PROPERTY boPin261_48XSFaultToolValue : BOOL
GET
                    boPin261_48XSFaultToolValue := boPin261_48XSFault.Value;

                  
END_GET
END_PROPERTY

PROPERTY boPin254_48XSFaultToolValue : BOOL
GET
                    boPin254_48XSFaultToolValue := boPin254_48XSFault.Value;

                  
END_GET
END_PROPERTY

PROPERTY boPin260_48XSFaultToolValue : BOOL
GET
                    boPin260_48XSFaultToolValue := boPin260_48XSFault.Value;

                  
END_GET
END_PROPERTY

PROPERTY boPin253_48XSFaultToolValue : BOOL
GET
                    boPin253_48XSFaultToolValue := boPin253_48XSFault.Value;

                  
END_GET
END_PROPERTY

PROPERTY boPin270_48XSFaultToolValue : BOOL
GET
                    boPin270_48XSFaultToolValue := boPin270_48XSFault.Value;

                  
END_GET
END_PROPERTY

PROPERTY boPin276_48XSFaultToolValue : BOOL
GET
                    boPin276_48XSFaultToolValue := boPin276_48XSFault.Value;

                  
END_GET
END_PROPERTY

PROPERTY boPin277_48XSFaultToolValue : BOOL
GET
                    boPin277_48XSFaultToolValue := boPin277_48XSFault.Value;

                  
END_GET
END_PROPERTY

PROPERTY boPin275_48XSFaultToolValue : BOOL
GET
                    boPin275_48XSFaultToolValue := boPin275_48XSFault.Value;

                  
END_GET
END_PROPERTY

PROPERTY boPin268_48XSFaultToolValue : BOOL
GET
                    boPin268_48XSFaultToolValue := boPin268_48XSFault.Value;

                  
END_GET
END_PROPERTY

PROPERTY boPin274_48XSFaultToolValue : BOOL
GET
                    boPin274_48XSFaultToolValue := boPin274_48XSFault.Value;

                  
END_GET
END_PROPERTY

PROPERTY boPin267_48XSFaultToolValue : BOOL
GET
                    boPin267_48XSFaultToolValue := boPin267_48XSFault.Value;

                  
END_GET
END_PROPERTY

METHOD InitializeCanSignals
                  boPin136_48XSFault.AppScalingDivisor :=1;
boPin136_48XSFault.AppScalingMultiplier :=1;
boPin136_48XSFault.AppScalingOffset :=0;
boPin136_48XSFault.AppUnit :="";
boPin136_48XSFault.CanDefault :=0;
boPin136_48XSFault.CanInit :=0;
boPin136_48XSFault.CanMax :=1;
boPin136_48XSFault.CanMin :=0;
boPin136_48XSFault.CanUnit :="";
boPin136_48XSFault.Description :="for the Neotec diag pages";
boPin136_48XSFault.ErrorReaction := eErrorReaction.ERSIG_DFLT;
boPin136_48XSFault.ReceiverAdress :=1;
boPin136_48XSFault.ToolScalingDivisor :=1;
boPin136_48XSFault.ToolScalingMultiplier :=1;
boPin136_48XSFault.ToolScalingOffset :=0;
boPin136_48XSFault.ToolUnit :="";

boPin148_48XSFault.AppScalingDivisor :=1;
boPin148_48XSFault.AppScalingMultiplier :=1;
boPin148_48XSFault.AppScalingOffset :=0;
boPin148_48XSFault.AppUnit :="";
boPin148_48XSFault.CanDefault :=0;
boPin148_48XSFault.CanInit :=0;
boPin148_48XSFault.CanMax :=1;
boPin148_48XSFault.CanMin :=0;
boPin148_48XSFault.CanUnit :="";
boPin148_48XSFault.Description :="for the Neotec diag pages";
boPin148_48XSFault.ErrorReaction := eErrorReaction.ERSIG_DFLT;
boPin148_48XSFault.ReceiverAdress :=1;
boPin148_48XSFault.ToolScalingDivisor :=1;
boPin148_48XSFault.ToolScalingMultiplier :=1;
boPin148_48XSFault.ToolScalingOffset :=0;
boPin148_48XSFault.ToolUnit :="";

boPin135_48XSFault.AppScalingDivisor :=1;
boPin135_48XSFault.AppScalingMultiplier :=1;
boPin135_48XSFault.AppScalingOffset :=0;
boPin135_48XSFault.AppUnit :="";
boPin135_48XSFault.CanDefault :=0;
boPin135_48XSFault.CanInit :=0;
boPin135_48XSFault.CanMax :=1;
boPin135_48XSFault.CanMin :=0;
boPin135_48XSFault.CanUnit :="";
boPin135_48XSFault.Description :="for the Neotec diag pages";
boPin135_48XSFault.ErrorReaction := eErrorReaction.ERSIG_DFLT;
boPin135_48XSFault.ReceiverAdress :=1;
boPin135_48XSFault.ToolScalingDivisor :=1;
boPin135_48XSFault.ToolScalingMultiplier :=1;
boPin135_48XSFault.ToolScalingOffset :=0;
boPin135_48XSFault.ToolUnit :="";

boPin147_48XSFault.AppScalingDivisor :=1;
boPin147_48XSFault.AppScalingMultiplier :=1;
boPin147_48XSFault.AppScalingOffset :=0;
boPin147_48XSFault.AppUnit :="";
boPin147_48XSFault.CanDefault :=0;
boPin147_48XSFault.CanInit :=0;
boPin147_48XSFault.CanMax :=1;
boPin147_48XSFault.CanMin :=0;
boPin147_48XSFault.CanUnit :="";
boPin147_48XSFault.Description :="for the Neotec diag pages";
boPin147_48XSFault.ErrorReaction := eErrorReaction.ERSIG_DFLT;
boPin147_48XSFault.ReceiverAdress :=1;
boPin147_48XSFault.ToolScalingDivisor :=1;
boPin147_48XSFault.ToolScalingMultiplier :=1;
boPin147_48XSFault.ToolScalingOffset :=0;
boPin147_48XSFault.ToolUnit :="";

boPin269_48XSFault.AppScalingDivisor :=1;
boPin269_48XSFault.AppScalingMultiplier :=1;
boPin269_48XSFault.AppScalingOffset :=0;
boPin269_48XSFault.AppUnit :="";
boPin269_48XSFault.CanDefault :=0;
boPin269_48XSFault.CanInit :=0;
boPin269_48XSFault.CanMax :=1;
boPin269_48XSFault.CanMin :=0;
boPin269_48XSFault.CanUnit :="";
boPin269_48XSFault.Description :="for the Neotec diag pages";
boPin269_48XSFault.ErrorReaction := eErrorReaction.ERSIG_DFLT;
boPin269_48XSFault.ReceiverAdress :=1;
boPin269_48XSFault.ToolScalingDivisor :=1;
boPin269_48XSFault.ToolScalingMultiplier :=1;
boPin269_48XSFault.ToolScalingOffset :=0;
boPin269_48XSFault.ToolUnit :="";

boPin118_48XSFault.AppScalingDivisor :=1;
boPin118_48XSFault.AppScalingMultiplier :=1;
boPin118_48XSFault.AppScalingOffset :=0;
boPin118_48XSFault.AppUnit :="";
boPin118_48XSFault.CanDefault :=0;
boPin118_48XSFault.CanInit :=0;
boPin118_48XSFault.CanMax :=1;
boPin118_48XSFault.CanMin :=0;
boPin118_48XSFault.CanUnit :="";
boPin118_48XSFault.Description :="for the Neotec diag pages";
boPin118_48XSFault.ErrorReaction := eErrorReaction.ERSIG_DFLT;
boPin118_48XSFault.ReceiverAdress :=1;
boPin118_48XSFault.ToolScalingDivisor :=1;
boPin118_48XSFault.ToolScalingMultiplier :=1;
boPin118_48XSFault.ToolScalingOffset :=0;
boPin118_48XSFault.ToolUnit :="";

boPin106_48XSFault.AppScalingDivisor :=1;
boPin106_48XSFault.AppScalingMultiplier :=1;
boPin106_48XSFault.AppScalingOffset :=0;
boPin106_48XSFault.AppUnit :="";
boPin106_48XSFault.CanDefault :=0;
boPin106_48XSFault.CanInit :=0;
boPin106_48XSFault.CanMax :=1;
boPin106_48XSFault.CanMin :=0;
boPin106_48XSFault.CanUnit :="";
boPin106_48XSFault.Description :="for the Neotec diag pages";
boPin106_48XSFault.ErrorReaction := eErrorReaction.ERSIG_DFLT;
boPin106_48XSFault.ReceiverAdress :=1;
boPin106_48XSFault.ToolScalingDivisor :=1;
boPin106_48XSFault.ToolScalingMultiplier :=1;
boPin106_48XSFault.ToolScalingOffset :=0;
boPin106_48XSFault.ToolUnit :="";

boPin117_48XSFault.AppScalingDivisor :=1;
boPin117_48XSFault.AppScalingMultiplier :=1;
boPin117_48XSFault.AppScalingOffset :=0;
boPin117_48XSFault.AppUnit :="";
boPin117_48XSFault.CanDefault :=0;
boPin117_48XSFault.CanInit :=0;
boPin117_48XSFault.CanMax :=1;
boPin117_48XSFault.CanMin :=0;
boPin117_48XSFault.CanUnit :="";
boPin117_48XSFault.Description :="for the Neotec diag pages";
boPin117_48XSFault.ErrorReaction := eErrorReaction.ERSIG_DFLT;
boPin117_48XSFault.ReceiverAdress :=1;
boPin117_48XSFault.ToolScalingDivisor :=1;
boPin117_48XSFault.ToolScalingMultiplier :=1;
boPin117_48XSFault.ToolScalingOffset :=0;
boPin117_48XSFault.ToolUnit :="";

boPin105_48XSFault.AppScalingDivisor :=1;
boPin105_48XSFault.AppScalingMultiplier :=1;
boPin105_48XSFault.AppScalingOffset :=0;
boPin105_48XSFault.AppUnit :="";
boPin105_48XSFault.CanDefault :=0;
boPin105_48XSFault.CanInit :=0;
boPin105_48XSFault.CanMax :=1;
boPin105_48XSFault.CanMin :=0;
boPin105_48XSFault.CanUnit :="";
boPin105_48XSFault.Description :="for the Neotec diag pages";
boPin105_48XSFault.ErrorReaction := eErrorReaction.ERSIG_DFLT;
boPin105_48XSFault.ReceiverAdress :=1;
boPin105_48XSFault.ToolScalingDivisor :=1;
boPin105_48XSFault.ToolScalingMultiplier :=1;
boPin105_48XSFault.ToolScalingOffset :=0;
boPin105_48XSFault.ToolUnit :="";

boPin116_48XSFault.AppScalingDivisor :=1;
boPin116_48XSFault.AppScalingMultiplier :=1;
boPin116_48XSFault.AppScalingOffset :=0;
boPin116_48XSFault.AppUnit :="";
boPin116_48XSFault.CanDefault :=0;
boPin116_48XSFault.CanInit :=0;
boPin116_48XSFault.CanMax :=1;
boPin116_48XSFault.CanMin :=0;
boPin116_48XSFault.CanUnit :="";
boPin116_48XSFault.Description :="for the Neotec diag pages";
boPin116_48XSFault.ErrorReaction := eErrorReaction.ERSIG_DFLT;
boPin116_48XSFault.ReceiverAdress :=1;
boPin116_48XSFault.ToolScalingDivisor :=1;
boPin116_48XSFault.ToolScalingMultiplier :=1;
boPin116_48XSFault.ToolScalingOffset :=0;
boPin116_48XSFault.ToolUnit :="";

boPin104_48XSFault.AppScalingDivisor :=1;
boPin104_48XSFault.AppScalingMultiplier :=1;
boPin104_48XSFault.AppScalingOffset :=0;
boPin104_48XSFault.AppUnit :="";
boPin104_48XSFault.CanDefault :=0;
boPin104_48XSFault.CanInit :=0;
boPin104_48XSFault.CanMax :=1;
boPin104_48XSFault.CanMin :=0;
boPin104_48XSFault.CanUnit :="";
boPin104_48XSFault.Description :="for the Neotec diag pages";
boPin104_48XSFault.ErrorReaction := eErrorReaction.ERSIG_DFLT;
boPin104_48XSFault.ReceiverAdress :=1;
boPin104_48XSFault.ToolScalingDivisor :=1;
boPin104_48XSFault.ToolScalingMultiplier :=1;
boPin104_48XSFault.ToolScalingOffset :=0;
boPin104_48XSFault.ToolUnit :="";

boPin115_48XSFault.AppScalingDivisor :=1;
boPin115_48XSFault.AppScalingMultiplier :=1;
boPin115_48XSFault.AppScalingOffset :=0;
boPin115_48XSFault.AppUnit :="";
boPin115_48XSFault.CanDefault :=0;
boPin115_48XSFault.CanInit :=0;
boPin115_48XSFault.CanMax :=1;
boPin115_48XSFault.CanMin :=0;
boPin115_48XSFault.CanUnit :="";
boPin115_48XSFault.Description :="for the Neotec diag pages";
boPin115_48XSFault.ErrorReaction := eErrorReaction.ERSIG_DFLT;
boPin115_48XSFault.ReceiverAdress :=1;
boPin115_48XSFault.ToolScalingDivisor :=1;
boPin115_48XSFault.ToolScalingMultiplier :=1;
boPin115_48XSFault.ToolScalingOffset :=0;
boPin115_48XSFault.ToolUnit :="";

boPin103_48XSFault.AppScalingDivisor :=1;
boPin103_48XSFault.AppScalingMultiplier :=1;
boPin103_48XSFault.AppScalingOffset :=0;
boPin103_48XSFault.AppUnit :="";
boPin103_48XSFault.CanDefault :=0;
boPin103_48XSFault.CanInit :=0;
boPin103_48XSFault.CanMax :=1;
boPin103_48XSFault.CanMin :=0;
boPin103_48XSFault.CanUnit :="";
boPin103_48XSFault.Description :="for the Neotec diag pages";
boPin103_48XSFault.ErrorReaction := eErrorReaction.ERSIG_DFLT;
boPin103_48XSFault.ReceiverAdress :=1;
boPin103_48XSFault.ToolScalingDivisor :=1;
boPin103_48XSFault.ToolScalingMultiplier :=1;
boPin103_48XSFault.ToolScalingOffset :=0;
boPin103_48XSFault.ToolUnit :="";

boPin120_48XSFault.AppScalingDivisor :=1;
boPin120_48XSFault.AppScalingMultiplier :=1;
boPin120_48XSFault.AppScalingOffset :=0;
boPin120_48XSFault.AppUnit :="";
boPin120_48XSFault.CanDefault :=0;
boPin120_48XSFault.CanInit :=0;
boPin120_48XSFault.CanMax :=1;
boPin120_48XSFault.CanMin :=0;
boPin120_48XSFault.CanUnit :="";
boPin120_48XSFault.Description :="for the Neotec diag pages";
boPin120_48XSFault.ErrorReaction := eErrorReaction.ERSIG_DFLT;
boPin120_48XSFault.ReceiverAdress :=1;
boPin120_48XSFault.ToolScalingDivisor :=1;
boPin120_48XSFault.ToolScalingMultiplier :=1;
boPin120_48XSFault.ToolScalingOffset :=0;
boPin120_48XSFault.ToolUnit :="";

boPin108_48XSFault.AppScalingDivisor :=1;
boPin108_48XSFault.AppScalingMultiplier :=1;
boPin108_48XSFault.AppScalingOffset :=0;
boPin108_48XSFault.AppUnit :="";
boPin108_48XSFault.CanDefault :=0;
boPin108_48XSFault.CanInit :=0;
boPin108_48XSFault.CanMax :=1;
boPin108_48XSFault.CanMin :=0;
boPin108_48XSFault.CanUnit :="";
boPin108_48XSFault.Description :="for the Neotec diag pages";
boPin108_48XSFault.ErrorReaction := eErrorReaction.ERSIG_DFLT;
boPin108_48XSFault.ReceiverAdress :=1;
boPin108_48XSFault.ToolScalingDivisor :=1;
boPin108_48XSFault.ToolScalingMultiplier :=1;
boPin108_48XSFault.ToolScalingOffset :=0;
boPin108_48XSFault.ToolUnit :="";

boPin119_48XSFault.AppScalingDivisor :=1;
boPin119_48XSFault.AppScalingMultiplier :=1;
boPin119_48XSFault.AppScalingOffset :=0;
boPin119_48XSFault.AppUnit :="";
boPin119_48XSFault.CanDefault :=0;
boPin119_48XSFault.CanInit :=0;
boPin119_48XSFault.CanMax :=1;
boPin119_48XSFault.CanMin :=0;
boPin119_48XSFault.CanUnit :="";
boPin119_48XSFault.Description :="for the Neotec diag pages";
boPin119_48XSFault.ErrorReaction := eErrorReaction.ERSIG_DFLT;
boPin119_48XSFault.ReceiverAdress :=1;
boPin119_48XSFault.ToolScalingDivisor :=1;
boPin119_48XSFault.ToolScalingMultiplier :=1;
boPin119_48XSFault.ToolScalingOffset :=0;
boPin119_48XSFault.ToolUnit :="";

boPin107_48XSFault.AppScalingDivisor :=1;
boPin107_48XSFault.AppScalingMultiplier :=1;
boPin107_48XSFault.AppScalingOffset :=0;
boPin107_48XSFault.AppUnit :="";
boPin107_48XSFault.CanDefault :=0;
boPin107_48XSFault.CanInit :=0;
boPin107_48XSFault.CanMax :=1;
boPin107_48XSFault.CanMin :=0;
boPin107_48XSFault.CanUnit :="";
boPin107_48XSFault.Description :="for the Neotec diag pages";
boPin107_48XSFault.ErrorReaction := eErrorReaction.ERSIG_DFLT;
boPin107_48XSFault.ReceiverAdress :=1;
boPin107_48XSFault.ToolScalingDivisor :=1;
boPin107_48XSFault.ToolScalingMultiplier :=1;
boPin107_48XSFault.ToolScalingOffset :=0;
boPin107_48XSFault.ToolUnit :="";

boPin144_48XSFault.AppScalingDivisor :=1;
boPin144_48XSFault.AppScalingMultiplier :=1;
boPin144_48XSFault.AppScalingOffset :=0;
boPin144_48XSFault.AppUnit :="";
boPin144_48XSFault.CanDefault :=0;
boPin144_48XSFault.CanInit :=0;
boPin144_48XSFault.CanMax :=1;
boPin144_48XSFault.CanMin :=0;
boPin144_48XSFault.CanUnit :="";
boPin144_48XSFault.Description :="for the Neotec diag pages";
boPin144_48XSFault.ErrorReaction := eErrorReaction.ERSIG_DFLT;
boPin144_48XSFault.ReceiverAdress :=1;
boPin144_48XSFault.ToolScalingDivisor :=1;
boPin144_48XSFault.ToolScalingMultiplier :=1;
boPin144_48XSFault.ToolScalingOffset :=0;
boPin144_48XSFault.ToolUnit :="";

boPin132_48XSFault.AppScalingDivisor :=1;
boPin132_48XSFault.AppScalingMultiplier :=1;
boPin132_48XSFault.AppScalingOffset :=0;
boPin132_48XSFault.AppUnit :="";
boPin132_48XSFault.CanDefault :=0;
boPin132_48XSFault.CanInit :=0;
boPin132_48XSFault.CanMax :=1;
boPin132_48XSFault.CanMin :=0;
boPin132_48XSFault.CanUnit :="";
boPin132_48XSFault.Description :="for the Neotec diag pages";
boPin132_48XSFault.ErrorReaction := eErrorReaction.ERSIG_DFLT;
boPin132_48XSFault.ReceiverAdress :=1;
boPin132_48XSFault.ToolScalingDivisor :=1;
boPin132_48XSFault.ToolScalingMultiplier :=1;
boPin132_48XSFault.ToolScalingOffset :=0;
boPin132_48XSFault.ToolUnit :="";

boPin143_48XSFault.AppScalingDivisor :=1;
boPin143_48XSFault.AppScalingMultiplier :=1;
boPin143_48XSFault.AppScalingOffset :=0;
boPin143_48XSFault.AppUnit :="";
boPin143_48XSFault.CanDefault :=0;
boPin143_48XSFault.CanInit :=0;
boPin143_48XSFault.CanMax :=1;
boPin143_48XSFault.CanMin :=0;
boPin143_48XSFault.CanUnit :="";
boPin143_48XSFault.Description :="for the Neotec diag pages";
boPin143_48XSFault.ErrorReaction := eErrorReaction.ERSIG_DFLT;
boPin143_48XSFault.ReceiverAdress :=1;
boPin143_48XSFault.ToolScalingDivisor :=1;
boPin143_48XSFault.ToolScalingMultiplier :=1;
boPin143_48XSFault.ToolScalingOffset :=0;
boPin143_48XSFault.ToolUnit :="";

boPin131_48XSFault.AppScalingDivisor :=1;
boPin131_48XSFault.AppScalingMultiplier :=1;
boPin131_48XSFault.AppScalingOffset :=0;
boPin131_48XSFault.AppUnit :="";
boPin131_48XSFault.CanDefault :=0;
boPin131_48XSFault.CanInit :=0;
boPin131_48XSFault.CanMax :=1;
boPin131_48XSFault.CanMin :=0;
boPin131_48XSFault.CanUnit :="";
boPin131_48XSFault.Description :="for the Neotec diag pages";
boPin131_48XSFault.ErrorReaction := eErrorReaction.ERSIG_DFLT;
boPin131_48XSFault.ReceiverAdress :=1;
boPin131_48XSFault.ToolScalingDivisor :=1;
boPin131_48XSFault.ToolScalingMultiplier :=1;
boPin131_48XSFault.ToolScalingOffset :=0;
boPin131_48XSFault.ToolUnit :="";

boPin142_48XSFault.AppScalingDivisor :=1;
boPin142_48XSFault.AppScalingMultiplier :=1;
boPin142_48XSFault.AppScalingOffset :=0;
boPin142_48XSFault.AppUnit :="";
boPin142_48XSFault.CanDefault :=0;
boPin142_48XSFault.CanInit :=0;
boPin142_48XSFault.CanMax :=1;
boPin142_48XSFault.CanMin :=0;
boPin142_48XSFault.CanUnit :="";
boPin142_48XSFault.Description :="for the Neotec diag pages";
boPin142_48XSFault.ErrorReaction := eErrorReaction.ERSIG_DFLT;
boPin142_48XSFault.ReceiverAdress :=1;
boPin142_48XSFault.ToolScalingDivisor :=1;
boPin142_48XSFault.ToolScalingMultiplier :=1;
boPin142_48XSFault.ToolScalingOffset :=0;
boPin142_48XSFault.ToolUnit :="";

boPin130_48XSFault.AppScalingDivisor :=1;
boPin130_48XSFault.AppScalingMultiplier :=1;
boPin130_48XSFault.AppScalingOffset :=0;
boPin130_48XSFault.AppUnit :="";
boPin130_48XSFault.CanDefault :=0;
boPin130_48XSFault.CanInit :=0;
boPin130_48XSFault.CanMax :=1;
boPin130_48XSFault.CanMin :=0;
boPin130_48XSFault.CanUnit :="";
boPin130_48XSFault.Description :="for the Neotec diag pages";
boPin130_48XSFault.ErrorReaction := eErrorReaction.ERSIG_DFLT;
boPin130_48XSFault.ReceiverAdress :=1;
boPin130_48XSFault.ToolScalingDivisor :=1;
boPin130_48XSFault.ToolScalingMultiplier :=1;
boPin130_48XSFault.ToolScalingOffset :=0;
boPin130_48XSFault.ToolUnit :="";

boPin141_48XSFault.AppScalingDivisor :=1;
boPin141_48XSFault.AppScalingMultiplier :=1;
boPin141_48XSFault.AppScalingOffset :=0;
boPin141_48XSFault.AppUnit :="";
boPin141_48XSFault.CanDefault :=0;
boPin141_48XSFault.CanInit :=0;
boPin141_48XSFault.CanMax :=1;
boPin141_48XSFault.CanMin :=0;
boPin141_48XSFault.CanUnit :="";
boPin141_48XSFault.Description :="for the Neotec diag pages";
boPin141_48XSFault.ErrorReaction := eErrorReaction.ERSIG_DFLT;
boPin141_48XSFault.ReceiverAdress :=1;
boPin141_48XSFault.ToolScalingDivisor :=1;
boPin141_48XSFault.ToolScalingMultiplier :=1;
boPin141_48XSFault.ToolScalingOffset :=0;
boPin141_48XSFault.ToolUnit :="";

boPin129_48XSFault.AppScalingDivisor :=1;
boPin129_48XSFault.AppScalingMultiplier :=1;
boPin129_48XSFault.AppScalingOffset :=0;
boPin129_48XSFault.AppUnit :="";
boPin129_48XSFault.CanDefault :=0;
boPin129_48XSFault.CanInit :=0;
boPin129_48XSFault.CanMax :=1;
boPin129_48XSFault.CanMin :=0;
boPin129_48XSFault.CanUnit :="";
boPin129_48XSFault.Description :="for the Neotec diag pages";
boPin129_48XSFault.ErrorReaction := eErrorReaction.ERSIG_DFLT;
boPin129_48XSFault.ReceiverAdress :=1;
boPin129_48XSFault.ToolScalingDivisor :=1;
boPin129_48XSFault.ToolScalingMultiplier :=1;
boPin129_48XSFault.ToolScalingOffset :=0;
boPin129_48XSFault.ToolUnit :="";

boPin152_48XSFault.AppScalingDivisor :=1;
boPin152_48XSFault.AppScalingMultiplier :=1;
boPin152_48XSFault.AppScalingOffset :=0;
boPin152_48XSFault.AppUnit :="";
boPin152_48XSFault.CanDefault :=0;
boPin152_48XSFault.CanInit :=0;
boPin152_48XSFault.CanMax :=1;
boPin152_48XSFault.CanMin :=0;
boPin152_48XSFault.CanUnit :="";
boPin152_48XSFault.Description :="for the Neotec diag pages";
boPin152_48XSFault.ErrorReaction := eErrorReaction.ERSIG_DFLT;
boPin152_48XSFault.ReceiverAdress :=1;
boPin152_48XSFault.ToolScalingDivisor :=1;
boPin152_48XSFault.ToolScalingMultiplier :=1;
boPin152_48XSFault.ToolScalingOffset :=0;
boPin152_48XSFault.ToolUnit :="";

boPin140_48XSFault.AppScalingDivisor :=1;
boPin140_48XSFault.AppScalingMultiplier :=1;
boPin140_48XSFault.AppScalingOffset :=0;
boPin140_48XSFault.AppUnit :="";
boPin140_48XSFault.CanDefault :=0;
boPin140_48XSFault.CanInit :=0;
boPin140_48XSFault.CanMax :=1;
boPin140_48XSFault.CanMin :=0;
boPin140_48XSFault.CanUnit :="";
boPin140_48XSFault.Description :="for the Neotec diag pages";
boPin140_48XSFault.ErrorReaction := eErrorReaction.ERSIG_DFLT;
boPin140_48XSFault.ReceiverAdress :=1;
boPin140_48XSFault.ToolScalingDivisor :=1;
boPin140_48XSFault.ToolScalingMultiplier :=1;
boPin140_48XSFault.ToolScalingOffset :=0;
boPin140_48XSFault.ToolUnit :="";

boPin151_48XSFault.AppScalingDivisor :=1;
boPin151_48XSFault.AppScalingMultiplier :=1;
boPin151_48XSFault.AppScalingOffset :=0;
boPin151_48XSFault.AppUnit :="";
boPin151_48XSFault.CanDefault :=0;
boPin151_48XSFault.CanInit :=0;
boPin151_48XSFault.CanMax :=1;
boPin151_48XSFault.CanMin :=0;
boPin151_48XSFault.CanUnit :="";
boPin151_48XSFault.Description :="for the Neotec diag pages";
boPin151_48XSFault.ErrorReaction := eErrorReaction.ERSIG_DFLT;
boPin151_48XSFault.ReceiverAdress :=1;
boPin151_48XSFault.ToolScalingDivisor :=1;
boPin151_48XSFault.ToolScalingMultiplier :=1;
boPin151_48XSFault.ToolScalingOffset :=0;
boPin151_48XSFault.ToolUnit :="";

boPin139_48XSFault.AppScalingDivisor :=1;
boPin139_48XSFault.AppScalingMultiplier :=1;
boPin139_48XSFault.AppScalingOffset :=0;
boPin139_48XSFault.AppUnit :="";
boPin139_48XSFault.CanDefault :=0;
boPin139_48XSFault.CanInit :=0;
boPin139_48XSFault.CanMax :=1;
boPin139_48XSFault.CanMin :=0;
boPin139_48XSFault.CanUnit :="";
boPin139_48XSFault.Description :="for the Neotec diag pages";
boPin139_48XSFault.ErrorReaction := eErrorReaction.ERSIG_DFLT;
boPin139_48XSFault.ReceiverAdress :=1;
boPin139_48XSFault.ToolScalingDivisor :=1;
boPin139_48XSFault.ToolScalingMultiplier :=1;
boPin139_48XSFault.ToolScalingOffset :=0;
boPin139_48XSFault.ToolUnit :="";

boPin150_48XSFault.AppScalingDivisor :=1;
boPin150_48XSFault.AppScalingMultiplier :=1;
boPin150_48XSFault.AppScalingOffset :=0;
boPin150_48XSFault.AppUnit :="";
boPin150_48XSFault.CanDefault :=0;
boPin150_48XSFault.CanInit :=0;
boPin150_48XSFault.CanMax :=1;
boPin150_48XSFault.CanMin :=0;
boPin150_48XSFault.CanUnit :="";
boPin150_48XSFault.Description :="for the Neotec diag pages";
boPin150_48XSFault.ErrorReaction := eErrorReaction.ERSIG_DFLT;
boPin150_48XSFault.ReceiverAdress :=1;
boPin150_48XSFault.ToolScalingDivisor :=1;
boPin150_48XSFault.ToolScalingMultiplier :=1;
boPin150_48XSFault.ToolScalingOffset :=0;
boPin150_48XSFault.ToolUnit :="";

boPin138_48XSFault.AppScalingDivisor :=1;
boPin138_48XSFault.AppScalingMultiplier :=1;
boPin138_48XSFault.AppScalingOffset :=0;
boPin138_48XSFault.AppUnit :="";
boPin138_48XSFault.CanDefault :=0;
boPin138_48XSFault.CanInit :=0;
boPin138_48XSFault.CanMax :=1;
boPin138_48XSFault.CanMin :=0;
boPin138_48XSFault.CanUnit :="";
boPin138_48XSFault.Description :="for the Neotec diag pages";
boPin138_48XSFault.ErrorReaction := eErrorReaction.ERSIG_DFLT;
boPin138_48XSFault.ReceiverAdress :=1;
boPin138_48XSFault.ToolScalingDivisor :=1;
boPin138_48XSFault.ToolScalingMultiplier :=1;
boPin138_48XSFault.ToolScalingOffset :=0;
boPin138_48XSFault.ToolUnit :="";

boPin149_48XSFault.AppScalingDivisor :=1;
boPin149_48XSFault.AppScalingMultiplier :=1;
boPin149_48XSFault.AppScalingOffset :=0;
boPin149_48XSFault.AppUnit :="";
boPin149_48XSFault.CanDefault :=0;
boPin149_48XSFault.CanInit :=0;
boPin149_48XSFault.CanMax :=1;
boPin149_48XSFault.CanMin :=0;
boPin149_48XSFault.CanUnit :="";
boPin149_48XSFault.Description :="for the Neotec diag pages";
boPin149_48XSFault.ErrorReaction := eErrorReaction.ERSIG_DFLT;
boPin149_48XSFault.ReceiverAdress :=1;
boPin149_48XSFault.ToolScalingDivisor :=1;
boPin149_48XSFault.ToolScalingMultiplier :=1;
boPin149_48XSFault.ToolScalingOffset :=0;
boPin149_48XSFault.ToolUnit :="";

boPin137_48XSFault.AppScalingDivisor :=1;
boPin137_48XSFault.AppScalingMultiplier :=1;
boPin137_48XSFault.AppScalingOffset :=0;
boPin137_48XSFault.AppUnit :="";
boPin137_48XSFault.CanDefault :=0;
boPin137_48XSFault.CanInit :=0;
boPin137_48XSFault.CanMax :=1;
boPin137_48XSFault.CanMin :=0;
boPin137_48XSFault.CanUnit :="";
boPin137_48XSFault.Description :="for the Neotec diag pages";
boPin137_48XSFault.ErrorReaction := eErrorReaction.ERSIG_DFLT;
boPin137_48XSFault.ReceiverAdress :=1;
boPin137_48XSFault.ToolScalingDivisor :=1;
boPin137_48XSFault.ToolScalingMultiplier :=1;
boPin137_48XSFault.ToolScalingOffset :=0;
boPin137_48XSFault.ToolUnit :="";

boPin126_48XSFault.AppScalingDivisor :=1;
boPin126_48XSFault.AppScalingMultiplier :=1;
boPin126_48XSFault.AppScalingOffset :=0;
boPin126_48XSFault.AppUnit :="";
boPin126_48XSFault.CanDefault :=0;
boPin126_48XSFault.CanInit :=0;
boPin126_48XSFault.CanMax :=1;
boPin126_48XSFault.CanMin :=0;
boPin126_48XSFault.CanUnit :="";
boPin126_48XSFault.Description :="for the Neotec diag pages";
boPin126_48XSFault.ErrorReaction := eErrorReaction.ERSIG_DFLT;
boPin126_48XSFault.ReceiverAdress :=1;
boPin126_48XSFault.ToolScalingDivisor :=1;
boPin126_48XSFault.ToolScalingMultiplier :=1;
boPin126_48XSFault.ToolScalingOffset :=0;
boPin126_48XSFault.ToolUnit :="";

boPin114_48XSFault.AppScalingDivisor :=1;
boPin114_48XSFault.AppScalingMultiplier :=1;
boPin114_48XSFault.AppScalingOffset :=0;
boPin114_48XSFault.AppUnit :="";
boPin114_48XSFault.CanDefault :=0;
boPin114_48XSFault.CanInit :=0;
boPin114_48XSFault.CanMax :=1;
boPin114_48XSFault.CanMin :=0;
boPin114_48XSFault.CanUnit :="";
boPin114_48XSFault.Description :="for the Neotec diag pages";
boPin114_48XSFault.ErrorReaction := eErrorReaction.ERSIG_DFLT;
boPin114_48XSFault.ReceiverAdress :=1;
boPin114_48XSFault.ToolScalingDivisor :=1;
boPin114_48XSFault.ToolScalingMultiplier :=1;
boPin114_48XSFault.ToolScalingOffset :=0;
boPin114_48XSFault.ToolUnit :="";

boPin125_48XSFault.AppScalingDivisor :=1;
boPin125_48XSFault.AppScalingMultiplier :=1;
boPin125_48XSFault.AppScalingOffset :=0;
boPin125_48XSFault.AppUnit :="";
boPin125_48XSFault.CanDefault :=0;
boPin125_48XSFault.CanInit :=0;
boPin125_48XSFault.CanMax :=1;
boPin125_48XSFault.CanMin :=0;
boPin125_48XSFault.CanUnit :="";
boPin125_48XSFault.Description :="for the Neotec diag pages";
boPin125_48XSFault.ErrorReaction := eErrorReaction.ERSIG_DFLT;
boPin125_48XSFault.ReceiverAdress :=1;
boPin125_48XSFault.ToolScalingDivisor :=1;
boPin125_48XSFault.ToolScalingMultiplier :=1;
boPin125_48XSFault.ToolScalingOffset :=0;
boPin125_48XSFault.ToolUnit :="";

boPin113_48XSFault.AppScalingDivisor :=1;
boPin113_48XSFault.AppScalingMultiplier :=1;
boPin113_48XSFault.AppScalingOffset :=0;
boPin113_48XSFault.AppUnit :="";
boPin113_48XSFault.CanDefault :=0;
boPin113_48XSFault.CanInit :=0;
boPin113_48XSFault.CanMax :=1;
boPin113_48XSFault.CanMin :=0;
boPin113_48XSFault.CanUnit :="";
boPin113_48XSFault.Description :="for the Neotec diag pages";
boPin113_48XSFault.ErrorReaction := eErrorReaction.ERSIG_DFLT;
boPin113_48XSFault.ReceiverAdress :=1;
boPin113_48XSFault.ToolScalingDivisor :=1;
boPin113_48XSFault.ToolScalingMultiplier :=1;
boPin113_48XSFault.ToolScalingOffset :=0;
boPin113_48XSFault.ToolUnit :="";

boPin124_48XSFault.AppScalingDivisor :=1;
boPin124_48XSFault.AppScalingMultiplier :=1;
boPin124_48XSFault.AppScalingOffset :=0;
boPin124_48XSFault.AppUnit :="";
boPin124_48XSFault.CanDefault :=0;
boPin124_48XSFault.CanInit :=0;
boPin124_48XSFault.CanMax :=1;
boPin124_48XSFault.CanMin :=0;
boPin124_48XSFault.CanUnit :="";
boPin124_48XSFault.Description :="for the Neotec diag pages";
boPin124_48XSFault.ErrorReaction := eErrorReaction.ERSIG_DFLT;
boPin124_48XSFault.ReceiverAdress :=1;
boPin124_48XSFault.ToolScalingDivisor :=1;
boPin124_48XSFault.ToolScalingMultiplier :=1;
boPin124_48XSFault.ToolScalingOffset :=0;
boPin124_48XSFault.ToolUnit :="";

boPin112_48XSFault.AppScalingDivisor :=1;
boPin112_48XSFault.AppScalingMultiplier :=1;
boPin112_48XSFault.AppScalingOffset :=0;
boPin112_48XSFault.AppUnit :="";
boPin112_48XSFault.CanDefault :=0;
boPin112_48XSFault.CanInit :=0;
boPin112_48XSFault.CanMax :=1;
boPin112_48XSFault.CanMin :=0;
boPin112_48XSFault.CanUnit :="";
boPin112_48XSFault.Description :="for the Neotec diag pages";
boPin112_48XSFault.ErrorReaction := eErrorReaction.ERSIG_DFLT;
boPin112_48XSFault.ReceiverAdress :=1;
boPin112_48XSFault.ToolScalingDivisor :=1;
boPin112_48XSFault.ToolScalingMultiplier :=1;
boPin112_48XSFault.ToolScalingOffset :=0;
boPin112_48XSFault.ToolUnit :="";

boPin123_48XSFault.AppScalingDivisor :=1;
boPin123_48XSFault.AppScalingMultiplier :=1;
boPin123_48XSFault.AppScalingOffset :=0;
boPin123_48XSFault.AppUnit :="";
boPin123_48XSFault.CanDefault :=0;
boPin123_48XSFault.CanInit :=0;
boPin123_48XSFault.CanMax :=1;
boPin123_48XSFault.CanMin :=0;
boPin123_48XSFault.CanUnit :="";
boPin123_48XSFault.Description :="for the Neotec diag pages";
boPin123_48XSFault.ErrorReaction := eErrorReaction.ERSIG_DFLT;
boPin123_48XSFault.ReceiverAdress :=1;
boPin123_48XSFault.ToolScalingDivisor :=1;
boPin123_48XSFault.ToolScalingMultiplier :=1;
boPin123_48XSFault.ToolScalingOffset :=0;
boPin123_48XSFault.ToolUnit :="";

boPin111_48XSFault.AppScalingDivisor :=1;
boPin111_48XSFault.AppScalingMultiplier :=1;
boPin111_48XSFault.AppScalingOffset :=0;
boPin111_48XSFault.AppUnit :="";
boPin111_48XSFault.CanDefault :=0;
boPin111_48XSFault.CanInit :=0;
boPin111_48XSFault.CanMax :=1;
boPin111_48XSFault.CanMin :=0;
boPin111_48XSFault.CanUnit :="";
boPin111_48XSFault.Description :="for the Neotec diag pages";
boPin111_48XSFault.ErrorReaction := eErrorReaction.ERSIG_DFLT;
boPin111_48XSFault.ReceiverAdress :=1;
boPin111_48XSFault.ToolScalingDivisor :=1;
boPin111_48XSFault.ToolScalingMultiplier :=1;
boPin111_48XSFault.ToolScalingOffset :=0;
boPin111_48XSFault.ToolUnit :="";

boPin133_48XSFault.AppScalingDivisor :=1;
boPin133_48XSFault.AppScalingMultiplier :=1;
boPin133_48XSFault.AppScalingOffset :=0;
boPin133_48XSFault.AppUnit :="";
boPin133_48XSFault.CanDefault :=0;
boPin133_48XSFault.CanInit :=0;
boPin133_48XSFault.CanMax :=1;
boPin133_48XSFault.CanMin :=0;
boPin133_48XSFault.CanUnit :="";
boPin133_48XSFault.Description :="for the Neotec diag pages";
boPin133_48XSFault.ErrorReaction := eErrorReaction.ERSIG_DFLT;
boPin133_48XSFault.ReceiverAdress :=1;
boPin133_48XSFault.ToolScalingDivisor :=1;
boPin133_48XSFault.ToolScalingMultiplier :=1;
boPin133_48XSFault.ToolScalingOffset :=0;
boPin133_48XSFault.ToolUnit :="";

boPin134_48XSFault.AppScalingDivisor :=1;
boPin134_48XSFault.AppScalingMultiplier :=1;
boPin134_48XSFault.AppScalingOffset :=0;
boPin134_48XSFault.AppUnit :="";
boPin134_48XSFault.CanDefault :=0;
boPin134_48XSFault.CanInit :=0;
boPin134_48XSFault.CanMax :=1;
boPin134_48XSFault.CanMin :=0;
boPin134_48XSFault.CanUnit :="";
boPin134_48XSFault.Description :="for the Neotec diag pages";
boPin134_48XSFault.ErrorReaction := eErrorReaction.ERSIG_DFLT;
boPin134_48XSFault.ReceiverAdress :=1;
boPin134_48XSFault.ToolScalingDivisor :=1;
boPin134_48XSFault.ToolScalingMultiplier :=1;
boPin134_48XSFault.ToolScalingOffset :=0;
boPin134_48XSFault.ToolUnit :="";

boPin145_48XSFault.AppScalingDivisor :=1;
boPin145_48XSFault.AppScalingMultiplier :=1;
boPin145_48XSFault.AppScalingOffset :=0;
boPin145_48XSFault.AppUnit :="";
boPin145_48XSFault.CanDefault :=0;
boPin145_48XSFault.CanInit :=0;
boPin145_48XSFault.CanMax :=1;
boPin145_48XSFault.CanMin :=0;
boPin145_48XSFault.CanUnit :="";
boPin145_48XSFault.Description :="for the Neotec diag pages";
boPin145_48XSFault.ErrorReaction := eErrorReaction.ERSIG_DFLT;
boPin145_48XSFault.ReceiverAdress :=1;
boPin145_48XSFault.ToolScalingDivisor :=1;
boPin145_48XSFault.ToolScalingMultiplier :=1;
boPin145_48XSFault.ToolScalingOffset :=0;
boPin145_48XSFault.ToolUnit :="";

boPin146_48XSFault.AppScalingDivisor :=1;
boPin146_48XSFault.AppScalingMultiplier :=1;
boPin146_48XSFault.AppScalingOffset :=0;
boPin146_48XSFault.AppUnit :="";
boPin146_48XSFault.CanDefault :=0;
boPin146_48XSFault.CanInit :=0;
boPin146_48XSFault.CanMax :=1;
boPin146_48XSFault.CanMin :=0;
boPin146_48XSFault.CanUnit :="";
boPin146_48XSFault.Description :="for the Neotec diag pages";
boPin146_48XSFault.ErrorReaction := eErrorReaction.ERSIG_DFLT;
boPin146_48XSFault.ReceiverAdress :=1;
boPin146_48XSFault.ToolScalingDivisor :=1;
boPin146_48XSFault.ToolScalingMultiplier :=1;
boPin146_48XSFault.ToolScalingOffset :=0;
boPin146_48XSFault.ToolUnit :="";

boPin263_48XSFault.AppScalingDivisor :=1;
boPin263_48XSFault.AppScalingMultiplier :=1;
boPin263_48XSFault.AppScalingOffset :=0;
boPin263_48XSFault.AppUnit :="";
boPin263_48XSFault.CanDefault :=0;
boPin263_48XSFault.CanInit :=0;
boPin263_48XSFault.CanMax :=1;
boPin263_48XSFault.CanMin :=0;
boPin263_48XSFault.CanUnit :="";
boPin263_48XSFault.Description :="for the Neotec diag pages";
boPin263_48XSFault.ErrorReaction := eErrorReaction.ERSIG_DFLT;
boPin263_48XSFault.ReceiverAdress :=1;
boPin263_48XSFault.ToolScalingDivisor :=1;
boPin263_48XSFault.ToolScalingMultiplier :=1;
boPin263_48XSFault.ToolScalingOffset :=0;
boPin263_48XSFault.ToolUnit :="";

boPin256_48XSFault.AppScalingDivisor :=1;
boPin256_48XSFault.AppScalingMultiplier :=1;
boPin256_48XSFault.AppScalingOffset :=0;
boPin256_48XSFault.AppUnit :="";
boPin256_48XSFault.CanDefault :=0;
boPin256_48XSFault.CanInit :=0;
boPin256_48XSFault.CanMax :=1;
boPin256_48XSFault.CanMin :=0;
boPin256_48XSFault.CanUnit :="";
boPin256_48XSFault.Description :="for the Neotec diag pages";
boPin256_48XSFault.ErrorReaction := eErrorReaction.ERSIG_DFLT;
boPin256_48XSFault.ReceiverAdress :=1;
boPin256_48XSFault.ToolScalingDivisor :=1;
boPin256_48XSFault.ToolScalingMultiplier :=1;
boPin256_48XSFault.ToolScalingOffset :=0;
boPin256_48XSFault.ToolUnit :="";

boPin262_48XSFault.AppScalingDivisor :=1;
boPin262_48XSFault.AppScalingMultiplier :=1;
boPin262_48XSFault.AppScalingOffset :=0;
boPin262_48XSFault.AppUnit :="";
boPin262_48XSFault.CanDefault :=0;
boPin262_48XSFault.CanInit :=0;
boPin262_48XSFault.CanMax :=1;
boPin262_48XSFault.CanMin :=0;
boPin262_48XSFault.CanUnit :="";
boPin262_48XSFault.Description :="for the Neotec diag pages";
boPin262_48XSFault.ErrorReaction := eErrorReaction.ERSIG_DFLT;
boPin262_48XSFault.ReceiverAdress :=1;
boPin262_48XSFault.ToolScalingDivisor :=1;
boPin262_48XSFault.ToolScalingMultiplier :=1;
boPin262_48XSFault.ToolScalingOffset :=0;
boPin262_48XSFault.ToolUnit :="";

boPin255_48XSFault.AppScalingDivisor :=1;
boPin255_48XSFault.AppScalingMultiplier :=1;
boPin255_48XSFault.AppScalingOffset :=0;
boPin255_48XSFault.AppUnit :="";
boPin255_48XSFault.CanDefault :=0;
boPin255_48XSFault.CanInit :=0;
boPin255_48XSFault.CanMax :=1;
boPin255_48XSFault.CanMin :=0;
boPin255_48XSFault.CanUnit :="";
boPin255_48XSFault.Description :="for the Neotec diag pages";
boPin255_48XSFault.ErrorReaction := eErrorReaction.ERSIG_DFLT;
boPin255_48XSFault.ReceiverAdress :=1;
boPin255_48XSFault.ToolScalingDivisor :=1;
boPin255_48XSFault.ToolScalingMultiplier :=1;
boPin255_48XSFault.ToolScalingOffset :=0;
boPin255_48XSFault.ToolUnit :="";

boPin261_48XSFault.AppScalingDivisor :=1;
boPin261_48XSFault.AppScalingMultiplier :=1;
boPin261_48XSFault.AppScalingOffset :=0;
boPin261_48XSFault.AppUnit :="";
boPin261_48XSFault.CanDefault :=0;
boPin261_48XSFault.CanInit :=0;
boPin261_48XSFault.CanMax :=1;
boPin261_48XSFault.CanMin :=0;
boPin261_48XSFault.CanUnit :="";
boPin261_48XSFault.Description :="for the Neotec diag pages";
boPin261_48XSFault.ErrorReaction := eErrorReaction.ERSIG_DFLT;
boPin261_48XSFault.ReceiverAdress :=1;
boPin261_48XSFault.ToolScalingDivisor :=1;
boPin261_48XSFault.ToolScalingMultiplier :=1;
boPin261_48XSFault.ToolScalingOffset :=0;
boPin261_48XSFault.ToolUnit :="";

boPin254_48XSFault.AppScalingDivisor :=1;
boPin254_48XSFault.AppScalingMultiplier :=1;
boPin254_48XSFault.AppScalingOffset :=0;
boPin254_48XSFault.AppUnit :="";
boPin254_48XSFault.CanDefault :=0;
boPin254_48XSFault.CanInit :=0;
boPin254_48XSFault.CanMax :=1;
boPin254_48XSFault.CanMin :=0;
boPin254_48XSFault.CanUnit :="";
boPin254_48XSFault.Description :="for the Neotec diag pages";
boPin254_48XSFault.ErrorReaction := eErrorReaction.ERSIG_DFLT;
boPin254_48XSFault.ReceiverAdress :=1;
boPin254_48XSFault.ToolScalingDivisor :=1;
boPin254_48XSFault.ToolScalingMultiplier :=1;
boPin254_48XSFault.ToolScalingOffset :=0;
boPin254_48XSFault.ToolUnit :="";

boPin260_48XSFault.AppScalingDivisor :=1;
boPin260_48XSFault.AppScalingMultiplier :=1;
boPin260_48XSFault.AppScalingOffset :=0;
boPin260_48XSFault.AppUnit :="";
boPin260_48XSFault.CanDefault :=0;
boPin260_48XSFault.CanInit :=0;
boPin260_48XSFault.CanMax :=1;
boPin260_48XSFault.CanMin :=0;
boPin260_48XSFault.CanUnit :="";
boPin260_48XSFault.Description :="for the Neotec diag pages";
boPin260_48XSFault.ErrorReaction := eErrorReaction.ERSIG_DFLT;
boPin260_48XSFault.ReceiverAdress :=1;
boPin260_48XSFault.ToolScalingDivisor :=1;
boPin260_48XSFault.ToolScalingMultiplier :=1;
boPin260_48XSFault.ToolScalingOffset :=0;
boPin260_48XSFault.ToolUnit :="";

boPin253_48XSFault.AppScalingDivisor :=1;
boPin253_48XSFault.AppScalingMultiplier :=1;
boPin253_48XSFault.AppScalingOffset :=0;
boPin253_48XSFault.AppUnit :="";
boPin253_48XSFault.CanDefault :=0;
boPin253_48XSFault.CanInit :=0;
boPin253_48XSFault.CanMax :=1;
boPin253_48XSFault.CanMin :=0;
boPin253_48XSFault.CanUnit :="";
boPin253_48XSFault.Description :="for the Neotec diag pages";
boPin253_48XSFault.ErrorReaction := eErrorReaction.ERSIG_DFLT;
boPin253_48XSFault.ReceiverAdress :=1;
boPin253_48XSFault.ToolScalingDivisor :=1;
boPin253_48XSFault.ToolScalingMultiplier :=1;
boPin253_48XSFault.ToolScalingOffset :=0;
boPin253_48XSFault.ToolUnit :="";

boPin270_48XSFault.AppScalingDivisor :=1;
boPin270_48XSFault.AppScalingMultiplier :=1;
boPin270_48XSFault.AppScalingOffset :=0;
boPin270_48XSFault.AppUnit :="";
boPin270_48XSFault.CanDefault :=0;
boPin270_48XSFault.CanInit :=0;
boPin270_48XSFault.CanMax :=1;
boPin270_48XSFault.CanMin :=0;
boPin270_48XSFault.CanUnit :="";
boPin270_48XSFault.Description :="for the Neotec diag pages";
boPin270_48XSFault.ErrorReaction := eErrorReaction.ERSIG_DFLT;
boPin270_48XSFault.ReceiverAdress :=1;
boPin270_48XSFault.ToolScalingDivisor :=1;
boPin270_48XSFault.ToolScalingMultiplier :=1;
boPin270_48XSFault.ToolScalingOffset :=0;
boPin270_48XSFault.ToolUnit :="";

boPin276_48XSFault.AppScalingDivisor :=1;
boPin276_48XSFault.AppScalingMultiplier :=1;
boPin276_48XSFault.AppScalingOffset :=0;
boPin276_48XSFault.AppUnit :="";
boPin276_48XSFault.CanDefault :=0;
boPin276_48XSFault.CanInit :=0;
boPin276_48XSFault.CanMax :=1;
boPin276_48XSFault.CanMin :=0;
boPin276_48XSFault.CanUnit :="";
boPin276_48XSFault.Description :="for the Neotec diag pages";
boPin276_48XSFault.ErrorReaction := eErrorReaction.ERSIG_DFLT;
boPin276_48XSFault.ReceiverAdress :=1;
boPin276_48XSFault.ToolScalingDivisor :=1;
boPin276_48XSFault.ToolScalingMultiplier :=1;
boPin276_48XSFault.ToolScalingOffset :=0;
boPin276_48XSFault.ToolUnit :="";

boPin277_48XSFault.AppScalingDivisor :=1;
boPin277_48XSFault.AppScalingMultiplier :=1;
boPin277_48XSFault.AppScalingOffset :=0;
boPin277_48XSFault.AppUnit :="";
boPin277_48XSFault.CanDefault :=0;
boPin277_48XSFault.CanInit :=0;
boPin277_48XSFault.CanMax :=1;
boPin277_48XSFault.CanMin :=0;
boPin277_48XSFault.CanUnit :="";
boPin277_48XSFault.Description :="for the Neotec diag pages";
boPin277_48XSFault.ErrorReaction := eErrorReaction.ERSIG_DFLT;
boPin277_48XSFault.ReceiverAdress :=1;
boPin277_48XSFault.ToolScalingDivisor :=1;
boPin277_48XSFault.ToolScalingMultiplier :=1;
boPin277_48XSFault.ToolScalingOffset :=0;
boPin277_48XSFault.ToolUnit :="";

boPin275_48XSFault.AppScalingDivisor :=1;
boPin275_48XSFault.AppScalingMultiplier :=1;
boPin275_48XSFault.AppScalingOffset :=0;
boPin275_48XSFault.AppUnit :="";
boPin275_48XSFault.CanDefault :=0;
boPin275_48XSFault.CanInit :=0;
boPin275_48XSFault.CanMax :=1;
boPin275_48XSFault.CanMin :=0;
boPin275_48XSFault.CanUnit :="";
boPin275_48XSFault.Description :="for the Neotec diag pages";
boPin275_48XSFault.ErrorReaction := eErrorReaction.ERSIG_DFLT;
boPin275_48XSFault.ReceiverAdress :=1;
boPin275_48XSFault.ToolScalingDivisor :=1;
boPin275_48XSFault.ToolScalingMultiplier :=1;
boPin275_48XSFault.ToolScalingOffset :=0;
boPin275_48XSFault.ToolUnit :="";

boPin268_48XSFault.AppScalingDivisor :=1;
boPin268_48XSFault.AppScalingMultiplier :=1;
boPin268_48XSFault.AppScalingOffset :=0;
boPin268_48XSFault.AppUnit :="";
boPin268_48XSFault.CanDefault :=0;
boPin268_48XSFault.CanInit :=0;
boPin268_48XSFault.CanMax :=1;
boPin268_48XSFault.CanMin :=0;
boPin268_48XSFault.CanUnit :="";
boPin268_48XSFault.Description :="for the Neotec diag pages";
boPin268_48XSFault.ErrorReaction := eErrorReaction.ERSIG_DFLT;
boPin268_48XSFault.ReceiverAdress :=1;
boPin268_48XSFault.ToolScalingDivisor :=1;
boPin268_48XSFault.ToolScalingMultiplier :=1;
boPin268_48XSFault.ToolScalingOffset :=0;
boPin268_48XSFault.ToolUnit :="";

boPin274_48XSFault.AppScalingDivisor :=1;
boPin274_48XSFault.AppScalingMultiplier :=1;
boPin274_48XSFault.AppScalingOffset :=0;
boPin274_48XSFault.AppUnit :="";
boPin274_48XSFault.CanDefault :=0;
boPin274_48XSFault.CanInit :=0;
boPin274_48XSFault.CanMax :=1;
boPin274_48XSFault.CanMin :=0;
boPin274_48XSFault.CanUnit :="";
boPin274_48XSFault.Description :="for the Neotec diag pages";
boPin274_48XSFault.ErrorReaction := eErrorReaction.ERSIG_DFLT;
boPin274_48XSFault.ReceiverAdress :=1;
boPin274_48XSFault.ToolScalingDivisor :=1;
boPin274_48XSFault.ToolScalingMultiplier :=1;
boPin274_48XSFault.ToolScalingOffset :=0;
boPin274_48XSFault.ToolUnit :="";

boPin267_48XSFault.AppScalingDivisor :=1;
boPin267_48XSFault.AppScalingMultiplier :=1;
boPin267_48XSFault.AppScalingOffset :=0;
boPin267_48XSFault.AppUnit :="";
boPin267_48XSFault.CanDefault :=0;
boPin267_48XSFault.CanInit :=0;
boPin267_48XSFault.CanMax :=1;
boPin267_48XSFault.CanMin :=0;
boPin267_48XSFault.CanUnit :="";
boPin267_48XSFault.Description :="for the Neotec diag pages";
boPin267_48XSFault.ErrorReaction := eErrorReaction.ERSIG_DFLT;
boPin267_48XSFault.ReceiverAdress :=1;
boPin267_48XSFault.ToolScalingDivisor :=1;
boPin267_48XSFault.ToolScalingMultiplier :=1;
boPin267_48XSFault.ToolScalingOffset :=0;
boPin267_48XSFault.ToolUnit :="";


                
END_METHOD
END_FUNCTION_BLOCK

FUNCTION_BLOCK Msg9C0SendToEvision7MessageClass EXTENDS CanReceiveMessageClass
  VAR_INPUT
    boPin144_48XS : BoolCanSignalClass;
    boPin132_48XS : BoolCanSignalClass;
    boPin143_48XS : BoolCanSignalClass;
    boPin131_48XS : BoolCanSignalClass;
    boPin142_48XS : BoolCanSignalClass;
    boPin130_48XS : BoolCanSignalClass;
    boPin141_48XS : BoolCanSignalClass;
    boPin129_48XS : BoolCanSignalClass;
    boPin152_48XS : BoolCanSignalClass;
    boPin140_48XS : BoolCanSignalClass;
    boPin151_48XS : BoolCanSignalClass;
    boPin139_48XS : BoolCanSignalClass;
    boPin150_48XS : BoolCanSignalClass;
    boPin138_48XS : BoolCanSignalClass;
    boPin149_48XS : BoolCanSignalClass;
    boPin263_48XS : BoolCanSignalClass;
    boPin256_48XS : BoolCanSignalClass;
    boPin262_48XS : BoolCanSignalClass;
    boPin255_48XS : BoolCanSignalClass;
    boPin261_48XS : BoolCanSignalClass;
    boPin254_48XS : BoolCanSignalClass;
    boPin260_48XS : BoolCanSignalClass;
    boPin253_48XS : BoolCanSignalClass;
    boPin275_48XS : BoolCanSignalClass;
    boPin268_48XS : BoolCanSignalClass;
    boPin274_48XS : BoolCanSignalClass;
    boPin267_48XS : BoolCanSignalClass;
    i16gPressureBrakeSensorValue : Int16CanSignalClass;
    u8gLightsMode : UInt8CanSignalClass;
    bogOsciServiceBrakinBrakeOn : BoolCanSignalClass;
    bogFixeServiceBrakinBrakeOn : BoolCanSignalClass;
    bogBothServiceBrakinBrakeOn : BoolCanSignalClass;
    bogActiveWhiteLights15746 : BoolCanSignalClass;
    Counter : UInt32CanSignalClass;
  END_VAR

            
          

METHOD SetData
  VAR_INPUT
    CanMsgPointer : POINTER TO CanMessageClass;
  END_VAR
                  IF IsValidPointer(canMsgPointer,'SetData') THEN
	SUPER^.SetData(CanMsgPointer);
	//Set the new data
	boPin144_48XS.Value := canMsgPointer^.GetBoolOnBit(0);
	boPin132_48XS.Value := canMsgPointer^.GetBoolOnBit(1);
	boPin143_48XS.Value := canMsgPointer^.GetBoolOnBit(2);
	boPin131_48XS.Value := canMsgPointer^.GetBoolOnBit(3);
	boPin142_48XS.Value := canMsgPointer^.GetBoolOnBit(4);
	boPin130_48XS.Value := canMsgPointer^.GetBoolOnBit(5);
	boPin141_48XS.Value := canMsgPointer^.GetBoolOnBit(6);
	boPin129_48XS.Value := canMsgPointer^.GetBoolOnBit(7);
	boPin152_48XS.Value := canMsgPointer^.GetBoolOnBit(8);
	boPin140_48XS.Value := canMsgPointer^.GetBoolOnBit(9);
	boPin151_48XS.Value := canMsgPointer^.GetBoolOnBit(10);
	boPin139_48XS.Value := canMsgPointer^.GetBoolOnBit(11);
	boPin150_48XS.Value := canMsgPointer^.GetBoolOnBit(12);
	boPin138_48XS.Value := canMsgPointer^.GetBoolOnBit(13);
	boPin149_48XS.Value := canMsgPointer^.GetBoolOnBit(14);
	boPin263_48XS.Value := canMsgPointer^.GetBoolOnBit(15);
	boPin256_48XS.Value := canMsgPointer^.GetBoolOnBit(16);
	boPin262_48XS.Value := canMsgPointer^.GetBoolOnBit(17);
	boPin255_48XS.Value := canMsgPointer^.GetBoolOnBit(18);
	boPin261_48XS.Value := canMsgPointer^.GetBoolOnBit(19);
	boPin254_48XS.Value := canMsgPointer^.GetBoolOnBit(20);
	boPin260_48XS.Value := canMsgPointer^.GetBoolOnBit(21);
	boPin253_48XS.Value := canMsgPointer^.GetBoolOnBit(22);
	boPin275_48XS.Value := canMsgPointer^.GetBoolOnBit(23);
	boPin268_48XS.Value := canMsgPointer^.GetBoolOnBit(24);
	boPin274_48XS.Value := canMsgPointer^.GetBoolOnBit(25);
	boPin267_48XS.Value := canMsgPointer^.GetBoolOnBit(26);
	i16gPressureBrakeSensorValue.Value := canMsgPointer^.GetInt16(32);
	u8gLightsMode.Value := canMsgPointer^.GetUint8(48);
	bogOsciServiceBrakinBrakeOn.Value := canMsgPointer^.GetBoolOnBit(56);
	bogFixeServiceBrakinBrakeOn.Value := canMsgPointer^.GetBoolOnBit(57);
	bogBothServiceBrakinBrakeOn.Value := canMsgPointer^.GetBoolOnBit(58);
	bogActiveWhiteLights15746.Value := canMsgPointer^.GetBoolOnBit(59);
	//And increase the counter
	Counter.Value := CanMsgPointer^.Counter.Value;
END_IF

                
END_METHOD

PROPERTY boPin144_48XSRawValue : BOOL
GET
                    boPin144_48XSRawValue := boPin144_48XS.Value;

                  
END_GET
END_PROPERTY

PROPERTY boPin132_48XSRawValue : BOOL
GET
                    boPin132_48XSRawValue := boPin132_48XS.Value;

                  
END_GET
END_PROPERTY

PROPERTY boPin143_48XSRawValue : BOOL
GET
                    boPin143_48XSRawValue := boPin143_48XS.Value;

                  
END_GET
END_PROPERTY

PROPERTY boPin131_48XSRawValue : BOOL
GET
                    boPin131_48XSRawValue := boPin131_48XS.Value;

                  
END_GET
END_PROPERTY

PROPERTY boPin142_48XSRawValue : BOOL
GET
                    boPin142_48XSRawValue := boPin142_48XS.Value;

                  
END_GET
END_PROPERTY

PROPERTY boPin130_48XSRawValue : BOOL
GET
                    boPin130_48XSRawValue := boPin130_48XS.Value;

                  
END_GET
END_PROPERTY

PROPERTY boPin141_48XSRawValue : BOOL
GET
                    boPin141_48XSRawValue := boPin141_48XS.Value;

                  
END_GET
END_PROPERTY

PROPERTY boPin129_48XSRawValue : BOOL
GET
                    boPin129_48XSRawValue := boPin129_48XS.Value;

                  
END_GET
END_PROPERTY

PROPERTY boPin152_48XSRawValue : BOOL
GET
                    boPin152_48XSRawValue := boPin152_48XS.Value;

                  
END_GET
END_PROPERTY

PROPERTY boPin140_48XSRawValue : BOOL
GET
                    boPin140_48XSRawValue := boPin140_48XS.Value;

                  
END_GET
END_PROPERTY

PROPERTY boPin151_48XSRawValue : BOOL
GET
                    boPin151_48XSRawValue := boPin151_48XS.Value;

                  
END_GET
END_PROPERTY

PROPERTY boPin139_48XSRawValue : BOOL
GET
                    boPin139_48XSRawValue := boPin139_48XS.Value;

                  
END_GET
END_PROPERTY

PROPERTY boPin150_48XSRawValue : BOOL
GET
                    boPin150_48XSRawValue := boPin150_48XS.Value;

                  
END_GET
END_PROPERTY

PROPERTY boPin138_48XSRawValue : BOOL
GET
                    boPin138_48XSRawValue := boPin138_48XS.Value;

                  
END_GET
END_PROPERTY

PROPERTY boPin149_48XSRawValue : BOOL
GET
                    boPin149_48XSRawValue := boPin149_48XS.Value;

                  
END_GET
END_PROPERTY

PROPERTY boPin263_48XSRawValue : BOOL
GET
                    boPin263_48XSRawValue := boPin263_48XS.Value;

                  
END_GET
END_PROPERTY

PROPERTY boPin256_48XSRawValue : BOOL
GET
                    boPin256_48XSRawValue := boPin256_48XS.Value;

                  
END_GET
END_PROPERTY

PROPERTY boPin262_48XSRawValue : BOOL
GET
                    boPin262_48XSRawValue := boPin262_48XS.Value;

                  
END_GET
END_PROPERTY

PROPERTY boPin255_48XSRawValue : BOOL
GET
                    boPin255_48XSRawValue := boPin255_48XS.Value;

                  
END_GET
END_PROPERTY

PROPERTY boPin261_48XSRawValue : BOOL
GET
                    boPin261_48XSRawValue := boPin261_48XS.Value;

                  
END_GET
END_PROPERTY

PROPERTY boPin254_48XSRawValue : BOOL
GET
                    boPin254_48XSRawValue := boPin254_48XS.Value;

                  
END_GET
END_PROPERTY

PROPERTY boPin260_48XSRawValue : BOOL
GET
                    boPin260_48XSRawValue := boPin260_48XS.Value;

                  
END_GET
END_PROPERTY

PROPERTY boPin253_48XSRawValue : BOOL
GET
                    boPin253_48XSRawValue := boPin253_48XS.Value;

                  
END_GET
END_PROPERTY

PROPERTY boPin275_48XSRawValue : BOOL
GET
                    boPin275_48XSRawValue := boPin275_48XS.Value;

                  
END_GET
END_PROPERTY

PROPERTY boPin268_48XSRawValue : BOOL
GET
                    boPin268_48XSRawValue := boPin268_48XS.Value;

                  
END_GET
END_PROPERTY

PROPERTY boPin274_48XSRawValue : BOOL
GET
                    boPin274_48XSRawValue := boPin274_48XS.Value;

                  
END_GET
END_PROPERTY

PROPERTY boPin267_48XSRawValue : BOOL
GET
                    boPin267_48XSRawValue := boPin267_48XS.Value;

                  
END_GET
END_PROPERTY

PROPERTY i16gPressureBrakeSensorValueRawValue : INT
GET
                    IF i16gPressureBrakeSensorValue.AppScalingMultiplier = 0 THEN
	_MatchLog^.Error("Get i16gPressureBrakeSensorValueRawValue", "Division by Zero!");
	RETURN;
End_IF

i16gPressureBrakeSensorValueRawValue := TO_INT((i16gPressureBrakeSensorValue.Value - i16gPressureBrakeSensorValue.AppScalingOffset) * i16gPressureBrakeSensorValue.AppScalingDivisor / i16gPressureBrakeSensorValue.AppScalingMultiplier);

                  
END_GET
END_PROPERTY

PROPERTY u8gLightsModeRawValue : USINT
GET
                    IF u8gLightsMode.AppScalingMultiplier = 0 THEN
	_MatchLog^.Error("Get u8gLightsModeRawValue", "Division by Zero!");
	RETURN;
End_IF

u8gLightsModeRawValue := TO_USINT((u8gLightsMode.Value - u8gLightsMode.AppScalingOffset) * u8gLightsMode.AppScalingDivisor / u8gLightsMode.AppScalingMultiplier);

                  
END_GET
END_PROPERTY

PROPERTY bogOsciServiceBrakinBrakeOnRawValue : BOOL
GET
                    bogOsciServiceBrakinBrakeOnRawValue := bogOsciServiceBrakinBrakeOn.Value;

                  
END_GET
END_PROPERTY

PROPERTY bogFixeServiceBrakinBrakeOnRawValue : BOOL
GET
                    bogFixeServiceBrakinBrakeOnRawValue := bogFixeServiceBrakinBrakeOn.Value;

                  
END_GET
END_PROPERTY

PROPERTY bogBothServiceBrakinBrakeOnRawValue : BOOL
GET
                    bogBothServiceBrakinBrakeOnRawValue := bogBothServiceBrakinBrakeOn.Value;

                  
END_GET
END_PROPERTY

PROPERTY bogActiveWhiteLights15746RawValue : BOOL
GET
                    bogActiveWhiteLights15746RawValue := bogActiveWhiteLights15746.Value;

                  
END_GET
END_PROPERTY

PROPERTY boPin144_48XSToolValue : BOOL
GET
                    boPin144_48XSToolValue := boPin144_48XS.Value;

                  
END_GET
END_PROPERTY

PROPERTY boPin132_48XSToolValue : BOOL
GET
                    boPin132_48XSToolValue := boPin132_48XS.Value;

                  
END_GET
END_PROPERTY

PROPERTY boPin143_48XSToolValue : BOOL
GET
                    boPin143_48XSToolValue := boPin143_48XS.Value;

                  
END_GET
END_PROPERTY

PROPERTY boPin131_48XSToolValue : BOOL
GET
                    boPin131_48XSToolValue := boPin131_48XS.Value;

                  
END_GET
END_PROPERTY

PROPERTY boPin142_48XSToolValue : BOOL
GET
                    boPin142_48XSToolValue := boPin142_48XS.Value;

                  
END_GET
END_PROPERTY

PROPERTY boPin130_48XSToolValue : BOOL
GET
                    boPin130_48XSToolValue := boPin130_48XS.Value;

                  
END_GET
END_PROPERTY

PROPERTY boPin141_48XSToolValue : BOOL
GET
                    boPin141_48XSToolValue := boPin141_48XS.Value;

                  
END_GET
END_PROPERTY

PROPERTY boPin129_48XSToolValue : BOOL
GET
                    boPin129_48XSToolValue := boPin129_48XS.Value;

                  
END_GET
END_PROPERTY

PROPERTY boPin152_48XSToolValue : BOOL
GET
                    boPin152_48XSToolValue := boPin152_48XS.Value;

                  
END_GET
END_PROPERTY

PROPERTY boPin140_48XSToolValue : BOOL
GET
                    boPin140_48XSToolValue := boPin140_48XS.Value;

                  
END_GET
END_PROPERTY

PROPERTY boPin151_48XSToolValue : BOOL
GET
                    boPin151_48XSToolValue := boPin151_48XS.Value;

                  
END_GET
END_PROPERTY

PROPERTY boPin139_48XSToolValue : BOOL
GET
                    boPin139_48XSToolValue := boPin139_48XS.Value;

                  
END_GET
END_PROPERTY

PROPERTY boPin150_48XSToolValue : BOOL
GET
                    boPin150_48XSToolValue := boPin150_48XS.Value;

                  
END_GET
END_PROPERTY

PROPERTY boPin138_48XSToolValue : BOOL
GET
                    boPin138_48XSToolValue := boPin138_48XS.Value;

                  
END_GET
END_PROPERTY

PROPERTY boPin149_48XSToolValue : BOOL
GET
                    boPin149_48XSToolValue := boPin149_48XS.Value;

                  
END_GET
END_PROPERTY

PROPERTY boPin263_48XSToolValue : BOOL
GET
                    boPin263_48XSToolValue := boPin263_48XS.Value;

                  
END_GET
END_PROPERTY

PROPERTY boPin256_48XSToolValue : BOOL
GET
                    boPin256_48XSToolValue := boPin256_48XS.Value;

                  
END_GET
END_PROPERTY

PROPERTY boPin262_48XSToolValue : BOOL
GET
                    boPin262_48XSToolValue := boPin262_48XS.Value;

                  
END_GET
END_PROPERTY

PROPERTY boPin255_48XSToolValue : BOOL
GET
                    boPin255_48XSToolValue := boPin255_48XS.Value;

                  
END_GET
END_PROPERTY

PROPERTY boPin261_48XSToolValue : BOOL
GET
                    boPin261_48XSToolValue := boPin261_48XS.Value;

                  
END_GET
END_PROPERTY

PROPERTY boPin254_48XSToolValue : BOOL
GET
                    boPin254_48XSToolValue := boPin254_48XS.Value;

                  
END_GET
END_PROPERTY

PROPERTY boPin260_48XSToolValue : BOOL
GET
                    boPin260_48XSToolValue := boPin260_48XS.Value;

                  
END_GET
END_PROPERTY

PROPERTY boPin253_48XSToolValue : BOOL
GET
                    boPin253_48XSToolValue := boPin253_48XS.Value;

                  
END_GET
END_PROPERTY

PROPERTY boPin275_48XSToolValue : BOOL
GET
                    boPin275_48XSToolValue := boPin275_48XS.Value;

                  
END_GET
END_PROPERTY

PROPERTY boPin268_48XSToolValue : BOOL
GET
                    boPin268_48XSToolValue := boPin268_48XS.Value;

                  
END_GET
END_PROPERTY

PROPERTY boPin274_48XSToolValue : BOOL
GET
                    boPin274_48XSToolValue := boPin274_48XS.Value;

                  
END_GET
END_PROPERTY

PROPERTY boPin267_48XSToolValue : BOOL
GET
                    boPin267_48XSToolValue := boPin267_48XS.Value;

                  
END_GET
END_PROPERTY

PROPERTY i16gPressureBrakeSensorValueToolValue : INT
GET
                    IF i16gPressureBrakeSensorValue.ToolScalingDivisor = 0 OR i16gPressureBrakeSensorValue.AppScalingMultiplier = 0 THEN
	_MatchLog^.Error("Get i16gPressureBrakeSensorValueToolValue", "Division by Zero!");
	RETURN;
END_IF

i16gPressureBrakeSensorValueToolValue := TO_INT(((i16gPressureBrakeSensorValue.Value - i16gPressureBrakeSensorValue.AppScalingOffset) * i16gPressureBrakeSensorValue.AppScalingDivisor / i16gPressureBrakeSensorValue.AppScalingMultiplier * i16gPressureBrakeSensorValue.ToolScalingMultiplier / i16gPressureBrakeSensorValue.ToolScalingDivisor) + i16gPressureBrakeSensorValue.ToolScalingOffset);

                  
END_GET
END_PROPERTY

PROPERTY u8gLightsModeToolValue : USINT
GET
                    IF u8gLightsMode.ToolScalingDivisor = 0 OR u8gLightsMode.AppScalingMultiplier = 0 THEN
	_MatchLog^.Error("Get u8gLightsModeToolValue", "Division by Zero!");
	RETURN;
END_IF

u8gLightsModeToolValue := TO_USINT(((u8gLightsMode.Value - u8gLightsMode.AppScalingOffset) * u8gLightsMode.AppScalingDivisor / u8gLightsMode.AppScalingMultiplier * u8gLightsMode.ToolScalingMultiplier / u8gLightsMode.ToolScalingDivisor) + u8gLightsMode.ToolScalingOffset);

                  
END_GET
END_PROPERTY

PROPERTY bogOsciServiceBrakinBrakeOnToolValue : BOOL
GET
                    bogOsciServiceBrakinBrakeOnToolValue := bogOsciServiceBrakinBrakeOn.Value;

                  
END_GET
END_PROPERTY

PROPERTY bogFixeServiceBrakinBrakeOnToolValue : BOOL
GET
                    bogFixeServiceBrakinBrakeOnToolValue := bogFixeServiceBrakinBrakeOn.Value;

                  
END_GET
END_PROPERTY

PROPERTY bogBothServiceBrakinBrakeOnToolValue : BOOL
GET
                    bogBothServiceBrakinBrakeOnToolValue := bogBothServiceBrakinBrakeOn.Value;

                  
END_GET
END_PROPERTY

PROPERTY bogActiveWhiteLights15746ToolValue : BOOL
GET
                    bogActiveWhiteLights15746ToolValue := bogActiveWhiteLights15746.Value;

                  
END_GET
END_PROPERTY

METHOD InitializeCanSignals
                  boPin144_48XS.AppScalingDivisor :=1;
boPin144_48XS.AppScalingMultiplier :=1;
boPin144_48XS.AppScalingOffset :=0;
boPin144_48XS.AppUnit :="";
boPin144_48XS.CanDefault :=0;
boPin144_48XS.CanInit :=0;
boPin144_48XS.CanMax :=1;
boPin144_48XS.CanMin :=0;
boPin144_48XS.CanUnit :="";
boPin144_48XS.Description :="for the Neotec diag pages";
boPin144_48XS.ErrorReaction := eErrorReaction.ERSIG_DFLT;
boPin144_48XS.ReceiverAdress :=1;
boPin144_48XS.ToolScalingDivisor :=1;
boPin144_48XS.ToolScalingMultiplier :=1;
boPin144_48XS.ToolScalingOffset :=0;
boPin144_48XS.ToolUnit :="";

boPin132_48XS.AppScalingDivisor :=1;
boPin132_48XS.AppScalingMultiplier :=1;
boPin132_48XS.AppScalingOffset :=0;
boPin132_48XS.AppUnit :="";
boPin132_48XS.CanDefault :=0;
boPin132_48XS.CanInit :=0;
boPin132_48XS.CanMax :=1;
boPin132_48XS.CanMin :=0;
boPin132_48XS.CanUnit :="";
boPin132_48XS.Description :="for the Neotec diag pages";
boPin132_48XS.ErrorReaction := eErrorReaction.ERSIG_DFLT;
boPin132_48XS.ReceiverAdress :=1;
boPin132_48XS.ToolScalingDivisor :=1;
boPin132_48XS.ToolScalingMultiplier :=1;
boPin132_48XS.ToolScalingOffset :=0;
boPin132_48XS.ToolUnit :="";

boPin143_48XS.AppScalingDivisor :=1;
boPin143_48XS.AppScalingMultiplier :=1;
boPin143_48XS.AppScalingOffset :=0;
boPin143_48XS.AppUnit :="";
boPin143_48XS.CanDefault :=0;
boPin143_48XS.CanInit :=0;
boPin143_48XS.CanMax :=1;
boPin143_48XS.CanMin :=0;
boPin143_48XS.CanUnit :="";
boPin143_48XS.Description :="for the Neotec diag pages";
boPin143_48XS.ErrorReaction := eErrorReaction.ERSIG_DFLT;
boPin143_48XS.ReceiverAdress :=1;
boPin143_48XS.ToolScalingDivisor :=1;
boPin143_48XS.ToolScalingMultiplier :=1;
boPin143_48XS.ToolScalingOffset :=0;
boPin143_48XS.ToolUnit :="";

boPin131_48XS.AppScalingDivisor :=1;
boPin131_48XS.AppScalingMultiplier :=1;
boPin131_48XS.AppScalingOffset :=0;
boPin131_48XS.AppUnit :="";
boPin131_48XS.CanDefault :=0;
boPin131_48XS.CanInit :=0;
boPin131_48XS.CanMax :=1;
boPin131_48XS.CanMin :=0;
boPin131_48XS.CanUnit :="";
boPin131_48XS.Description :="for the Neotec diag pages";
boPin131_48XS.ErrorReaction := eErrorReaction.ERSIG_DFLT;
boPin131_48XS.ReceiverAdress :=1;
boPin131_48XS.ToolScalingDivisor :=1;
boPin131_48XS.ToolScalingMultiplier :=1;
boPin131_48XS.ToolScalingOffset :=0;
boPin131_48XS.ToolUnit :="";

boPin142_48XS.AppScalingDivisor :=1;
boPin142_48XS.AppScalingMultiplier :=1;
boPin142_48XS.AppScalingOffset :=0;
boPin142_48XS.AppUnit :="";
boPin142_48XS.CanDefault :=0;
boPin142_48XS.CanInit :=0;
boPin142_48XS.CanMax :=1;
boPin142_48XS.CanMin :=0;
boPin142_48XS.CanUnit :="";
boPin142_48XS.Description :="for the Neotec diag pages";
boPin142_48XS.ErrorReaction := eErrorReaction.ERSIG_DFLT;
boPin142_48XS.ReceiverAdress :=1;
boPin142_48XS.ToolScalingDivisor :=1;
boPin142_48XS.ToolScalingMultiplier :=1;
boPin142_48XS.ToolScalingOffset :=0;
boPin142_48XS.ToolUnit :="";

boPin130_48XS.AppScalingDivisor :=1;
boPin130_48XS.AppScalingMultiplier :=1;
boPin130_48XS.AppScalingOffset :=0;
boPin130_48XS.AppUnit :="";
boPin130_48XS.CanDefault :=0;
boPin130_48XS.CanInit :=0;
boPin130_48XS.CanMax :=1;
boPin130_48XS.CanMin :=0;
boPin130_48XS.CanUnit :="";
boPin130_48XS.Description :="for the Neotec diag pages";
boPin130_48XS.ErrorReaction := eErrorReaction.ERSIG_DFLT;
boPin130_48XS.ReceiverAdress :=1;
boPin130_48XS.ToolScalingDivisor :=1;
boPin130_48XS.ToolScalingMultiplier :=1;
boPin130_48XS.ToolScalingOffset :=0;
boPin130_48XS.ToolUnit :="";

boPin141_48XS.AppScalingDivisor :=1;
boPin141_48XS.AppScalingMultiplier :=1;
boPin141_48XS.AppScalingOffset :=0;
boPin141_48XS.AppUnit :="";
boPin141_48XS.CanDefault :=0;
boPin141_48XS.CanInit :=0;
boPin141_48XS.CanMax :=1;
boPin141_48XS.CanMin :=0;
boPin141_48XS.CanUnit :="";
boPin141_48XS.Description :="for the Neotec diag pages";
boPin141_48XS.ErrorReaction := eErrorReaction.ERSIG_DFLT;
boPin141_48XS.ReceiverAdress :=1;
boPin141_48XS.ToolScalingDivisor :=1;
boPin141_48XS.ToolScalingMultiplier :=1;
boPin141_48XS.ToolScalingOffset :=0;
boPin141_48XS.ToolUnit :="";

boPin129_48XS.AppScalingDivisor :=1;
boPin129_48XS.AppScalingMultiplier :=1;
boPin129_48XS.AppScalingOffset :=0;
boPin129_48XS.AppUnit :="";
boPin129_48XS.CanDefault :=0;
boPin129_48XS.CanInit :=0;
boPin129_48XS.CanMax :=1;
boPin129_48XS.CanMin :=0;
boPin129_48XS.CanUnit :="";
boPin129_48XS.Description :="for the Neotec diag pages";
boPin129_48XS.ErrorReaction := eErrorReaction.ERSIG_DFLT;
boPin129_48XS.ReceiverAdress :=1;
boPin129_48XS.ToolScalingDivisor :=1;
boPin129_48XS.ToolScalingMultiplier :=1;
boPin129_48XS.ToolScalingOffset :=0;
boPin129_48XS.ToolUnit :="";

boPin152_48XS.AppScalingDivisor :=1;
boPin152_48XS.AppScalingMultiplier :=1;
boPin152_48XS.AppScalingOffset :=0;
boPin152_48XS.AppUnit :="";
boPin152_48XS.CanDefault :=0;
boPin152_48XS.CanInit :=0;
boPin152_48XS.CanMax :=1;
boPin152_48XS.CanMin :=0;
boPin152_48XS.CanUnit :="";
boPin152_48XS.Description :="for the Neotec diag pages";
boPin152_48XS.ErrorReaction := eErrorReaction.ERSIG_DFLT;
boPin152_48XS.ReceiverAdress :=1;
boPin152_48XS.ToolScalingDivisor :=1;
boPin152_48XS.ToolScalingMultiplier :=1;
boPin152_48XS.ToolScalingOffset :=0;
boPin152_48XS.ToolUnit :="";

boPin140_48XS.AppScalingDivisor :=1;
boPin140_48XS.AppScalingMultiplier :=1;
boPin140_48XS.AppScalingOffset :=0;
boPin140_48XS.AppUnit :="";
boPin140_48XS.CanDefault :=0;
boPin140_48XS.CanInit :=0;
boPin140_48XS.CanMax :=1;
boPin140_48XS.CanMin :=0;
boPin140_48XS.CanUnit :="";
boPin140_48XS.Description :="for the Neotec diag pages";
boPin140_48XS.ErrorReaction := eErrorReaction.ERSIG_DFLT;
boPin140_48XS.ReceiverAdress :=1;
boPin140_48XS.ToolScalingDivisor :=1;
boPin140_48XS.ToolScalingMultiplier :=1;
boPin140_48XS.ToolScalingOffset :=0;
boPin140_48XS.ToolUnit :="";

boPin151_48XS.AppScalingDivisor :=1;
boPin151_48XS.AppScalingMultiplier :=1;
boPin151_48XS.AppScalingOffset :=0;
boPin151_48XS.AppUnit :="";
boPin151_48XS.CanDefault :=0;
boPin151_48XS.CanInit :=0;
boPin151_48XS.CanMax :=1;
boPin151_48XS.CanMin :=0;
boPin151_48XS.CanUnit :="";
boPin151_48XS.Description :="for the Neotec diag pages";
boPin151_48XS.ErrorReaction := eErrorReaction.ERSIG_DFLT;
boPin151_48XS.ReceiverAdress :=1;
boPin151_48XS.ToolScalingDivisor :=1;
boPin151_48XS.ToolScalingMultiplier :=1;
boPin151_48XS.ToolScalingOffset :=0;
boPin151_48XS.ToolUnit :="";

boPin139_48XS.AppScalingDivisor :=1;
boPin139_48XS.AppScalingMultiplier :=1;
boPin139_48XS.AppScalingOffset :=0;
boPin139_48XS.AppUnit :="";
boPin139_48XS.CanDefault :=0;
boPin139_48XS.CanInit :=0;
boPin139_48XS.CanMax :=1;
boPin139_48XS.CanMin :=0;
boPin139_48XS.CanUnit :="";
boPin139_48XS.Description :="for the Neotec diag pages";
boPin139_48XS.ErrorReaction := eErrorReaction.ERSIG_DFLT;
boPin139_48XS.ReceiverAdress :=1;
boPin139_48XS.ToolScalingDivisor :=1;
boPin139_48XS.ToolScalingMultiplier :=1;
boPin139_48XS.ToolScalingOffset :=0;
boPin139_48XS.ToolUnit :="";

boPin150_48XS.AppScalingDivisor :=1;
boPin150_48XS.AppScalingMultiplier :=1;
boPin150_48XS.AppScalingOffset :=0;
boPin150_48XS.AppUnit :="";
boPin150_48XS.CanDefault :=0;
boPin150_48XS.CanInit :=0;
boPin150_48XS.CanMax :=1;
boPin150_48XS.CanMin :=0;
boPin150_48XS.CanUnit :="";
boPin150_48XS.Description :="for the Neotec diag pages";
boPin150_48XS.ErrorReaction := eErrorReaction.ERSIG_DFLT;
boPin150_48XS.ReceiverAdress :=1;
boPin150_48XS.ToolScalingDivisor :=1;
boPin150_48XS.ToolScalingMultiplier :=1;
boPin150_48XS.ToolScalingOffset :=0;
boPin150_48XS.ToolUnit :="";

boPin138_48XS.AppScalingDivisor :=1;
boPin138_48XS.AppScalingMultiplier :=1;
boPin138_48XS.AppScalingOffset :=0;
boPin138_48XS.AppUnit :="";
boPin138_48XS.CanDefault :=0;
boPin138_48XS.CanInit :=0;
boPin138_48XS.CanMax :=1;
boPin138_48XS.CanMin :=0;
boPin138_48XS.CanUnit :="";
boPin138_48XS.Description :="for the Neotec diag pages";
boPin138_48XS.ErrorReaction := eErrorReaction.ERSIG_DFLT;
boPin138_48XS.ReceiverAdress :=1;
boPin138_48XS.ToolScalingDivisor :=1;
boPin138_48XS.ToolScalingMultiplier :=1;
boPin138_48XS.ToolScalingOffset :=0;
boPin138_48XS.ToolUnit :="";

boPin149_48XS.AppScalingDivisor :=1;
boPin149_48XS.AppScalingMultiplier :=1;
boPin149_48XS.AppScalingOffset :=0;
boPin149_48XS.AppUnit :="";
boPin149_48XS.CanDefault :=0;
boPin149_48XS.CanInit :=0;
boPin149_48XS.CanMax :=1;
boPin149_48XS.CanMin :=0;
boPin149_48XS.CanUnit :="";
boPin149_48XS.Description :="for the Neotec diag pages";
boPin149_48XS.ErrorReaction := eErrorReaction.ERSIG_DFLT;
boPin149_48XS.ReceiverAdress :=1;
boPin149_48XS.ToolScalingDivisor :=1;
boPin149_48XS.ToolScalingMultiplier :=1;
boPin149_48XS.ToolScalingOffset :=0;
boPin149_48XS.ToolUnit :="";

boPin263_48XS.AppScalingDivisor :=1;
boPin263_48XS.AppScalingMultiplier :=1;
boPin263_48XS.AppScalingOffset :=0;
boPin263_48XS.AppUnit :="";
boPin263_48XS.CanDefault :=0;
boPin263_48XS.CanInit :=0;
boPin263_48XS.CanMax :=1;
boPin263_48XS.CanMin :=0;
boPin263_48XS.CanUnit :="";
boPin263_48XS.Description :="for the Neotec diag pages";
boPin263_48XS.ErrorReaction := eErrorReaction.ERSIG_DFLT;
boPin263_48XS.ReceiverAdress :=1;
boPin263_48XS.ToolScalingDivisor :=1;
boPin263_48XS.ToolScalingMultiplier :=1;
boPin263_48XS.ToolScalingOffset :=0;
boPin263_48XS.ToolUnit :="";

boPin256_48XS.AppScalingDivisor :=1;
boPin256_48XS.AppScalingMultiplier :=1;
boPin256_48XS.AppScalingOffset :=0;
boPin256_48XS.AppUnit :="";
boPin256_48XS.CanDefault :=0;
boPin256_48XS.CanInit :=0;
boPin256_48XS.CanMax :=1;
boPin256_48XS.CanMin :=0;
boPin256_48XS.CanUnit :="";
boPin256_48XS.Description :="for the Neotec diag pages";
boPin256_48XS.ErrorReaction := eErrorReaction.ERSIG_DFLT;
boPin256_48XS.ReceiverAdress :=1;
boPin256_48XS.ToolScalingDivisor :=1;
boPin256_48XS.ToolScalingMultiplier :=1;
boPin256_48XS.ToolScalingOffset :=0;
boPin256_48XS.ToolUnit :="";

boPin262_48XS.AppScalingDivisor :=1;
boPin262_48XS.AppScalingMultiplier :=1;
boPin262_48XS.AppScalingOffset :=0;
boPin262_48XS.AppUnit :="";
boPin262_48XS.CanDefault :=0;
boPin262_48XS.CanInit :=0;
boPin262_48XS.CanMax :=1;
boPin262_48XS.CanMin :=0;
boPin262_48XS.CanUnit :="";
boPin262_48XS.Description :="for the Neotec diag pages";
boPin262_48XS.ErrorReaction := eErrorReaction.ERSIG_DFLT;
boPin262_48XS.ReceiverAdress :=1;
boPin262_48XS.ToolScalingDivisor :=1;
boPin262_48XS.ToolScalingMultiplier :=1;
boPin262_48XS.ToolScalingOffset :=0;
boPin262_48XS.ToolUnit :="";

boPin255_48XS.AppScalingDivisor :=1;
boPin255_48XS.AppScalingMultiplier :=1;
boPin255_48XS.AppScalingOffset :=0;
boPin255_48XS.AppUnit :="";
boPin255_48XS.CanDefault :=0;
boPin255_48XS.CanInit :=0;
boPin255_48XS.CanMax :=1;
boPin255_48XS.CanMin :=0;
boPin255_48XS.CanUnit :="";
boPin255_48XS.Description :="for the Neotec diag pages";
boPin255_48XS.ErrorReaction := eErrorReaction.ERSIG_DFLT;
boPin255_48XS.ReceiverAdress :=1;
boPin255_48XS.ToolScalingDivisor :=1;
boPin255_48XS.ToolScalingMultiplier :=1;
boPin255_48XS.ToolScalingOffset :=0;
boPin255_48XS.ToolUnit :="";

boPin261_48XS.AppScalingDivisor :=1;
boPin261_48XS.AppScalingMultiplier :=1;
boPin261_48XS.AppScalingOffset :=0;
boPin261_48XS.AppUnit :="";
boPin261_48XS.CanDefault :=0;
boPin261_48XS.CanInit :=0;
boPin261_48XS.CanMax :=1;
boPin261_48XS.CanMin :=0;
boPin261_48XS.CanUnit :="";
boPin261_48XS.Description :="for the Neotec diag pages";
boPin261_48XS.ErrorReaction := eErrorReaction.ERSIG_DFLT;
boPin261_48XS.ReceiverAdress :=1;
boPin261_48XS.ToolScalingDivisor :=1;
boPin261_48XS.ToolScalingMultiplier :=1;
boPin261_48XS.ToolScalingOffset :=0;
boPin261_48XS.ToolUnit :="";

boPin254_48XS.AppScalingDivisor :=1;
boPin254_48XS.AppScalingMultiplier :=1;
boPin254_48XS.AppScalingOffset :=0;
boPin254_48XS.AppUnit :="";
boPin254_48XS.CanDefault :=0;
boPin254_48XS.CanInit :=0;
boPin254_48XS.CanMax :=1;
boPin254_48XS.CanMin :=0;
boPin254_48XS.CanUnit :="";
boPin254_48XS.Description :="for the Neotec diag pages";
boPin254_48XS.ErrorReaction := eErrorReaction.ERSIG_DFLT;
boPin254_48XS.ReceiverAdress :=1;
boPin254_48XS.ToolScalingDivisor :=1;
boPin254_48XS.ToolScalingMultiplier :=1;
boPin254_48XS.ToolScalingOffset :=0;
boPin254_48XS.ToolUnit :="";

boPin260_48XS.AppScalingDivisor :=1;
boPin260_48XS.AppScalingMultiplier :=1;
boPin260_48XS.AppScalingOffset :=0;
boPin260_48XS.AppUnit :="";
boPin260_48XS.CanDefault :=0;
boPin260_48XS.CanInit :=0;
boPin260_48XS.CanMax :=1;
boPin260_48XS.CanMin :=0;
boPin260_48XS.CanUnit :="";
boPin260_48XS.Description :="for the Neotec diag pages";
boPin260_48XS.ErrorReaction := eErrorReaction.ERSIG_DFLT;
boPin260_48XS.ReceiverAdress :=1;
boPin260_48XS.ToolScalingDivisor :=1;
boPin260_48XS.ToolScalingMultiplier :=1;
boPin260_48XS.ToolScalingOffset :=0;
boPin260_48XS.ToolUnit :="";

boPin253_48XS.AppScalingDivisor :=1;
boPin253_48XS.AppScalingMultiplier :=1;
boPin253_48XS.AppScalingOffset :=0;
boPin253_48XS.AppUnit :="";
boPin253_48XS.CanDefault :=0;
boPin253_48XS.CanInit :=0;
boPin253_48XS.CanMax :=1;
boPin253_48XS.CanMin :=0;
boPin253_48XS.CanUnit :="";
boPin253_48XS.Description :="for the Neotec diag pages";
boPin253_48XS.ErrorReaction := eErrorReaction.ERSIG_DFLT;
boPin253_48XS.ReceiverAdress :=1;
boPin253_48XS.ToolScalingDivisor :=1;
boPin253_48XS.ToolScalingMultiplier :=1;
boPin253_48XS.ToolScalingOffset :=0;
boPin253_48XS.ToolUnit :="";

boPin275_48XS.AppScalingDivisor :=1;
boPin275_48XS.AppScalingMultiplier :=1;
boPin275_48XS.AppScalingOffset :=0;
boPin275_48XS.AppUnit :="";
boPin275_48XS.CanDefault :=0;
boPin275_48XS.CanInit :=0;
boPin275_48XS.CanMax :=1;
boPin275_48XS.CanMin :=0;
boPin275_48XS.CanUnit :="";
boPin275_48XS.Description :="for the Neotec diag pages";
boPin275_48XS.ErrorReaction := eErrorReaction.ERSIG_DFLT;
boPin275_48XS.ReceiverAdress :=1;
boPin275_48XS.ToolScalingDivisor :=1;
boPin275_48XS.ToolScalingMultiplier :=1;
boPin275_48XS.ToolScalingOffset :=0;
boPin275_48XS.ToolUnit :="";

boPin268_48XS.AppScalingDivisor :=1;
boPin268_48XS.AppScalingMultiplier :=1;
boPin268_48XS.AppScalingOffset :=0;
boPin268_48XS.AppUnit :="";
boPin268_48XS.CanDefault :=0;
boPin268_48XS.CanInit :=0;
boPin268_48XS.CanMax :=1;
boPin268_48XS.CanMin :=0;
boPin268_48XS.CanUnit :="";
boPin268_48XS.Description :="for the Neotec diag pages";
boPin268_48XS.ErrorReaction := eErrorReaction.ERSIG_DFLT;
boPin268_48XS.ReceiverAdress :=1;
boPin268_48XS.ToolScalingDivisor :=1;
boPin268_48XS.ToolScalingMultiplier :=1;
boPin268_48XS.ToolScalingOffset :=0;
boPin268_48XS.ToolUnit :="";

boPin274_48XS.AppScalingDivisor :=1;
boPin274_48XS.AppScalingMultiplier :=1;
boPin274_48XS.AppScalingOffset :=0;
boPin274_48XS.AppUnit :="";
boPin274_48XS.CanDefault :=0;
boPin274_48XS.CanInit :=0;
boPin274_48XS.CanMax :=1;
boPin274_48XS.CanMin :=0;
boPin274_48XS.CanUnit :="";
boPin274_48XS.Description :="for the Neotec diag pages";
boPin274_48XS.ErrorReaction := eErrorReaction.ERSIG_DFLT;
boPin274_48XS.ReceiverAdress :=1;
boPin274_48XS.ToolScalingDivisor :=1;
boPin274_48XS.ToolScalingMultiplier :=1;
boPin274_48XS.ToolScalingOffset :=0;
boPin274_48XS.ToolUnit :="";

boPin267_48XS.AppScalingDivisor :=1;
boPin267_48XS.AppScalingMultiplier :=1;
boPin267_48XS.AppScalingOffset :=0;
boPin267_48XS.AppUnit :="";
boPin267_48XS.CanDefault :=0;
boPin267_48XS.CanInit :=0;
boPin267_48XS.CanMax :=1;
boPin267_48XS.CanMin :=0;
boPin267_48XS.CanUnit :="";
boPin267_48XS.Description :="for the Neotec diag pages";
boPin267_48XS.ErrorReaction := eErrorReaction.ERSIG_DFLT;
boPin267_48XS.ReceiverAdress :=1;
boPin267_48XS.ToolScalingDivisor :=1;
boPin267_48XS.ToolScalingMultiplier :=1;
boPin267_48XS.ToolScalingOffset :=0;
boPin267_48XS.ToolUnit :="";

i16gPressureBrakeSensorValue.AppScalingDivisor :=1;
i16gPressureBrakeSensorValue.AppScalingMultiplier :=1;
i16gPressureBrakeSensorValue.AppScalingOffset :=0;
i16gPressureBrakeSensorValue.AppUnit :="";
i16gPressureBrakeSensorValue.CanDefault :=0;
i16gPressureBrakeSensorValue.CanInit :=0;
i16gPressureBrakeSensorValue.CanMax :=VBasic.LibConst.I16_MAX;
i16gPressureBrakeSensorValue.CanMin :=VBasic.LibConst.I16_MIN;
i16gPressureBrakeSensorValue.CanUnit :="";
i16gPressureBrakeSensorValue.Description :="for the Neotec diag pages";
i16gPressureBrakeSensorValue.ErrorReaction := eErrorReaction.ERSIG_DFLT;
i16gPressureBrakeSensorValue.ReceiverAdress :=1;
i16gPressureBrakeSensorValue.ToolScalingDivisor :=1;
i16gPressureBrakeSensorValue.ToolScalingMultiplier :=1;
i16gPressureBrakeSensorValue.ToolScalingOffset :=0;
i16gPressureBrakeSensorValue.ToolUnit :="";

u8gLightsMode.AppScalingDivisor :=1;
u8gLightsMode.AppScalingMultiplier :=1;
u8gLightsMode.AppScalingOffset :=0;
u8gLightsMode.AppUnit :="";
u8gLightsMode.CanDefault :=0;
u8gLightsMode.CanInit :=0;
u8gLightsMode.CanMax :=VBasic.LibConst.U8_MAX;
u8gLightsMode.CanMin :=VBasic.LibConst.U8_MIN;
u8gLightsMode.CanUnit :="";
u8gLightsMode.Description :="for the Neotec diag pages";
u8gLightsMode.ErrorReaction := eErrorReaction.ERSIG_DFLT;
u8gLightsMode.ReceiverAdress :=1;
u8gLightsMode.ToolScalingDivisor :=1;
u8gLightsMode.ToolScalingMultiplier :=1;
u8gLightsMode.ToolScalingOffset :=0;
u8gLightsMode.ToolUnit :="";

bogOsciServiceBrakinBrakeOn.AppScalingDivisor :=1;
bogOsciServiceBrakinBrakeOn.AppScalingMultiplier :=1;
bogOsciServiceBrakinBrakeOn.AppScalingOffset :=0;
bogOsciServiceBrakinBrakeOn.AppUnit :="";
bogOsciServiceBrakinBrakeOn.CanDefault :=0;
bogOsciServiceBrakinBrakeOn.CanInit :=0;
bogOsciServiceBrakinBrakeOn.CanMax :=1;
bogOsciServiceBrakinBrakeOn.CanMin :=0;
bogOsciServiceBrakinBrakeOn.CanUnit :="";
bogOsciServiceBrakinBrakeOn.Description :="Activation rodage frein essieu oscillant";
bogOsciServiceBrakinBrakeOn.ErrorReaction := eErrorReaction.ERSIG_DFLT;
bogOsciServiceBrakinBrakeOn.ReceiverAdress :=1;
bogOsciServiceBrakinBrakeOn.ToolScalingDivisor :=1;
bogOsciServiceBrakinBrakeOn.ToolScalingMultiplier :=1;
bogOsciServiceBrakinBrakeOn.ToolScalingOffset :=0;
bogOsciServiceBrakinBrakeOn.ToolUnit :="";

bogFixeServiceBrakinBrakeOn.AppScalingDivisor :=1;
bogFixeServiceBrakinBrakeOn.AppScalingMultiplier :=1;
bogFixeServiceBrakinBrakeOn.AppScalingOffset :=0;
bogFixeServiceBrakinBrakeOn.AppUnit :="";
bogFixeServiceBrakinBrakeOn.CanDefault :=0;
bogFixeServiceBrakinBrakeOn.CanInit :=0;
bogFixeServiceBrakinBrakeOn.CanMax :=1;
bogFixeServiceBrakinBrakeOn.CanMin :=0;
bogFixeServiceBrakinBrakeOn.CanUnit :="";
bogFixeServiceBrakinBrakeOn.Description :="Activation rodage frein essieu fixe";
bogFixeServiceBrakinBrakeOn.ErrorReaction := eErrorReaction.ERSIG_DFLT;
bogFixeServiceBrakinBrakeOn.ReceiverAdress :=1;
bogFixeServiceBrakinBrakeOn.ToolScalingDivisor :=1;
bogFixeServiceBrakinBrakeOn.ToolScalingMultiplier :=1;
bogFixeServiceBrakinBrakeOn.ToolScalingOffset :=0;
bogFixeServiceBrakinBrakeOn.ToolUnit :="";

bogBothServiceBrakinBrakeOn.AppScalingDivisor :=1;
bogBothServiceBrakinBrakeOn.AppScalingMultiplier :=1;
bogBothServiceBrakinBrakeOn.AppScalingOffset :=0;
bogBothServiceBrakinBrakeOn.AppUnit :="";
bogBothServiceBrakinBrakeOn.CanDefault :=0;
bogBothServiceBrakinBrakeOn.CanInit :=0;
bogBothServiceBrakinBrakeOn.CanMax :=1;
bogBothServiceBrakinBrakeOn.CanMin :=0;
bogBothServiceBrakinBrakeOn.CanUnit :="";
bogBothServiceBrakinBrakeOn.Description :="Activation rodage deux freins";
bogBothServiceBrakinBrakeOn.ErrorReaction := eErrorReaction.ERSIG_DFLT;
bogBothServiceBrakinBrakeOn.ReceiverAdress :=1;
bogBothServiceBrakinBrakeOn.ToolScalingDivisor :=1;
bogBothServiceBrakinBrakeOn.ToolScalingMultiplier :=1;
bogBothServiceBrakinBrakeOn.ToolScalingOffset :=0;
bogBothServiceBrakinBrakeOn.ToolUnit :="";

bogActiveWhiteLights15746.AppScalingDivisor :=1;
bogActiveWhiteLights15746.AppScalingMultiplier :=1;
bogActiveWhiteLights15746.AppScalingOffset :=0;
bogActiveWhiteLights15746.AppUnit :="";
bogActiveWhiteLights15746.CanDefault :=0;
bogActiveWhiteLights15746.CanInit :=0;
bogActiveWhiteLights15746.CanMax :=1;
bogActiveWhiteLights15746.CanMin :=0;
bogActiveWhiteLights15746.CanUnit :="";
bogActiveWhiteLights15746.Description :="new signal";
bogActiveWhiteLights15746.ErrorReaction := eErrorReaction.ERSIG_DFLT;
bogActiveWhiteLights15746.ReceiverAdress :=1;
bogActiveWhiteLights15746.ToolScalingDivisor :=1;
bogActiveWhiteLights15746.ToolScalingMultiplier :=1;
bogActiveWhiteLights15746.ToolScalingOffset :=0;
bogActiveWhiteLights15746.ToolUnit :="";


                
END_METHOD
END_FUNCTION_BLOCK

FUNCTION_BLOCK Msg10C0SendToEvision7MessageClass EXTENDS CanReceiveMessageClass
  VAR_INPUT
    i16gPressureBlockOscillation : Int16CanSignalClass;
    u8gTTC580Version_Major : UInt8CanSignalClass;
    u8gTTC580Version_Minor : UInt8CanSignalClass;
    u8gTTC580Version_Patch : UInt8CanSignalClass;
    u8gTTC580Version_Custom : UInt8CanSignalClass;
    i16gJoystAdvanceScaling : Int16CanSignalClass;
    Counter : UInt32CanSignalClass;
  END_VAR

            
          

METHOD SetData
  VAR_INPUT
    CanMsgPointer : POINTER TO CanMessageClass;
  END_VAR
                  IF IsValidPointer(canMsgPointer,'SetData') THEN
	SUPER^.SetData(CanMsgPointer);
	//Set the new data
	i16gPressureBlockOscillation.Value := canMsgPointer^.GetInt16(0);
	u8gTTC580Version_Major.Value := canMsgPointer^.GetUint8(16);
	u8gTTC580Version_Minor.Value := canMsgPointer^.GetUint8(24);
	u8gTTC580Version_Patch.Value := canMsgPointer^.GetUint8(32);
	u8gTTC580Version_Custom.Value := canMsgPointer^.GetUint8(40);
	i16gJoystAdvanceScaling.Value := canMsgPointer^.GetInt16(48);
	//And increase the counter
	Counter.Value := CanMsgPointer^.Counter.Value;
END_IF

                
END_METHOD

PROPERTY i16gPressureBlockOscillationRawValue : INT
GET
                    IF i16gPressureBlockOscillation.AppScalingMultiplier = 0 THEN
	_MatchLog^.Error("Get i16gPressureBlockOscillationRawValue", "Division by Zero!");
	RETURN;
End_IF

i16gPressureBlockOscillationRawValue := TO_INT((i16gPressureBlockOscillation.Value - i16gPressureBlockOscillation.AppScalingOffset) * i16gPressureBlockOscillation.AppScalingDivisor / i16gPressureBlockOscillation.AppScalingMultiplier);

                  
END_GET
END_PROPERTY

PROPERTY u8gTTC580Version_MajorRawValue : USINT
GET
                    IF u8gTTC580Version_Major.AppScalingMultiplier = 0 THEN
	_MatchLog^.Error("Get u8gTTC580Version_MajorRawValue", "Division by Zero!");
	RETURN;
End_IF

u8gTTC580Version_MajorRawValue := TO_USINT((u8gTTC580Version_Major.Value - u8gTTC580Version_Major.AppScalingOffset) * u8gTTC580Version_Major.AppScalingDivisor / u8gTTC580Version_Major.AppScalingMultiplier);

                  
END_GET
END_PROPERTY

PROPERTY u8gTTC580Version_MinorRawValue : USINT
GET
                    IF u8gTTC580Version_Minor.AppScalingMultiplier = 0 THEN
	_MatchLog^.Error("Get u8gTTC580Version_MinorRawValue", "Division by Zero!");
	RETURN;
End_IF

u8gTTC580Version_MinorRawValue := TO_USINT((u8gTTC580Version_Minor.Value - u8gTTC580Version_Minor.AppScalingOffset) * u8gTTC580Version_Minor.AppScalingDivisor / u8gTTC580Version_Minor.AppScalingMultiplier);

                  
END_GET
END_PROPERTY

PROPERTY u8gTTC580Version_PatchRawValue : USINT
GET
                    IF u8gTTC580Version_Patch.AppScalingMultiplier = 0 THEN
	_MatchLog^.Error("Get u8gTTC580Version_PatchRawValue", "Division by Zero!");
	RETURN;
End_IF

u8gTTC580Version_PatchRawValue := TO_USINT((u8gTTC580Version_Patch.Value - u8gTTC580Version_Patch.AppScalingOffset) * u8gTTC580Version_Patch.AppScalingDivisor / u8gTTC580Version_Patch.AppScalingMultiplier);

                  
END_GET
END_PROPERTY

PROPERTY u8gTTC580Version_CustomRawValue : USINT
GET
                    IF u8gTTC580Version_Custom.AppScalingMultiplier = 0 THEN
	_MatchLog^.Error("Get u8gTTC580Version_CustomRawValue", "Division by Zero!");
	RETURN;
End_IF

u8gTTC580Version_CustomRawValue := TO_USINT((u8gTTC580Version_Custom.Value - u8gTTC580Version_Custom.AppScalingOffset) * u8gTTC580Version_Custom.AppScalingDivisor / u8gTTC580Version_Custom.AppScalingMultiplier);

                  
END_GET
END_PROPERTY

PROPERTY i16gJoystAdvanceScalingRawValue : INT
GET
                    IF i16gJoystAdvanceScaling.AppScalingMultiplier = 0 THEN
	_MatchLog^.Error("Get i16gJoystAdvanceScalingRawValue", "Division by Zero!");
	RETURN;
End_IF

i16gJoystAdvanceScalingRawValue := TO_INT((i16gJoystAdvanceScaling.Value - i16gJoystAdvanceScaling.AppScalingOffset) * i16gJoystAdvanceScaling.AppScalingDivisor / i16gJoystAdvanceScaling.AppScalingMultiplier);

                  
END_GET
END_PROPERTY

PROPERTY i16gPressureBlockOscillationToolValue : INT
GET
                    IF i16gPressureBlockOscillation.ToolScalingDivisor = 0 OR i16gPressureBlockOscillation.AppScalingMultiplier = 0 THEN
	_MatchLog^.Error("Get i16gPressureBlockOscillationToolValue", "Division by Zero!");
	RETURN;
END_IF

i16gPressureBlockOscillationToolValue := TO_INT(((i16gPressureBlockOscillation.Value - i16gPressureBlockOscillation.AppScalingOffset) * i16gPressureBlockOscillation.AppScalingDivisor / i16gPressureBlockOscillation.AppScalingMultiplier * i16gPressureBlockOscillation.ToolScalingMultiplier / i16gPressureBlockOscillation.ToolScalingDivisor) + i16gPressureBlockOscillation.ToolScalingOffset);

                  
END_GET
END_PROPERTY

PROPERTY u8gTTC580Version_MajorToolValue : USINT
GET
                    IF u8gTTC580Version_Major.ToolScalingDivisor = 0 OR u8gTTC580Version_Major.AppScalingMultiplier = 0 THEN
	_MatchLog^.Error("Get u8gTTC580Version_MajorToolValue", "Division by Zero!");
	RETURN;
END_IF

u8gTTC580Version_MajorToolValue := TO_USINT(((u8gTTC580Version_Major.Value - u8gTTC580Version_Major.AppScalingOffset) * u8gTTC580Version_Major.AppScalingDivisor / u8gTTC580Version_Major.AppScalingMultiplier * u8gTTC580Version_Major.ToolScalingMultiplier / u8gTTC580Version_Major.ToolScalingDivisor) + u8gTTC580Version_Major.ToolScalingOffset);

                  
END_GET
END_PROPERTY

PROPERTY u8gTTC580Version_MinorToolValue : USINT
GET
                    IF u8gTTC580Version_Minor.ToolScalingDivisor = 0 OR u8gTTC580Version_Minor.AppScalingMultiplier = 0 THEN
	_MatchLog^.Error("Get u8gTTC580Version_MinorToolValue", "Division by Zero!");
	RETURN;
END_IF

u8gTTC580Version_MinorToolValue := TO_USINT(((u8gTTC580Version_Minor.Value - u8gTTC580Version_Minor.AppScalingOffset) * u8gTTC580Version_Minor.AppScalingDivisor / u8gTTC580Version_Minor.AppScalingMultiplier * u8gTTC580Version_Minor.ToolScalingMultiplier / u8gTTC580Version_Minor.ToolScalingDivisor) + u8gTTC580Version_Minor.ToolScalingOffset);

                  
END_GET
END_PROPERTY

PROPERTY u8gTTC580Version_PatchToolValue : USINT
GET
                    IF u8gTTC580Version_Patch.ToolScalingDivisor = 0 OR u8gTTC580Version_Patch.AppScalingMultiplier = 0 THEN
	_MatchLog^.Error("Get u8gTTC580Version_PatchToolValue", "Division by Zero!");
	RETURN;
END_IF

u8gTTC580Version_PatchToolValue := TO_USINT(((u8gTTC580Version_Patch.Value - u8gTTC580Version_Patch.AppScalingOffset) * u8gTTC580Version_Patch.AppScalingDivisor / u8gTTC580Version_Patch.AppScalingMultiplier * u8gTTC580Version_Patch.ToolScalingMultiplier / u8gTTC580Version_Patch.ToolScalingDivisor) + u8gTTC580Version_Patch.ToolScalingOffset);

                  
END_GET
END_PROPERTY

PROPERTY u8gTTC580Version_CustomToolValue : USINT
GET
                    IF u8gTTC580Version_Custom.ToolScalingDivisor = 0 OR u8gTTC580Version_Custom.AppScalingMultiplier = 0 THEN
	_MatchLog^.Error("Get u8gTTC580Version_CustomToolValue", "Division by Zero!");
	RETURN;
END_IF

u8gTTC580Version_CustomToolValue := TO_USINT(((u8gTTC580Version_Custom.Value - u8gTTC580Version_Custom.AppScalingOffset) * u8gTTC580Version_Custom.AppScalingDivisor / u8gTTC580Version_Custom.AppScalingMultiplier * u8gTTC580Version_Custom.ToolScalingMultiplier / u8gTTC580Version_Custom.ToolScalingDivisor) + u8gTTC580Version_Custom.ToolScalingOffset);

                  
END_GET
END_PROPERTY

PROPERTY i16gJoystAdvanceScalingToolValue : INT
GET
                    IF i16gJoystAdvanceScaling.ToolScalingDivisor = 0 OR i16gJoystAdvanceScaling.AppScalingMultiplier = 0 THEN
	_MatchLog^.Error("Get i16gJoystAdvanceScalingToolValue", "Division by Zero!");
	RETURN;
END_IF

i16gJoystAdvanceScalingToolValue := TO_INT(((i16gJoystAdvanceScaling.Value - i16gJoystAdvanceScaling.AppScalingOffset) * i16gJoystAdvanceScaling.AppScalingDivisor / i16gJoystAdvanceScaling.AppScalingMultiplier * i16gJoystAdvanceScaling.ToolScalingMultiplier / i16gJoystAdvanceScaling.ToolScalingDivisor) + i16gJoystAdvanceScaling.ToolScalingOffset);

                  
END_GET
END_PROPERTY

METHOD InitializeCanSignals
                  i16gPressureBlockOscillation.AppScalingDivisor :=1;
i16gPressureBlockOscillation.AppScalingMultiplier :=1;
i16gPressureBlockOscillation.AppScalingOffset :=0;
i16gPressureBlockOscillation.AppUnit :="";
i16gPressureBlockOscillation.CanDefault :=0;
i16gPressureBlockOscillation.CanInit :=0;
i16gPressureBlockOscillation.CanMax :=VBasic.LibConst.I16_MAX;
i16gPressureBlockOscillation.CanMin :=VBasic.LibConst.I16_MIN;
i16gPressureBlockOscillation.CanUnit :="";
i16gPressureBlockOscillation.Description :="Oscillation block pressure";
i16gPressureBlockOscillation.ErrorReaction := eErrorReaction.ERSIG_DFLT;
i16gPressureBlockOscillation.ReceiverAdress :=1;
i16gPressureBlockOscillation.ToolScalingDivisor :=1;
i16gPressureBlockOscillation.ToolScalingMultiplier :=1;
i16gPressureBlockOscillation.ToolScalingOffset :=0;
i16gPressureBlockOscillation.ToolUnit :="";

u8gTTC580Version_Major.AppScalingDivisor :=1;
u8gTTC580Version_Major.AppScalingMultiplier :=1;
u8gTTC580Version_Major.AppScalingOffset :=0;
u8gTTC580Version_Major.AppUnit :="";
u8gTTC580Version_Major.CanDefault :=0;
u8gTTC580Version_Major.CanInit :=0;
u8gTTC580Version_Major.CanMax :=VBasic.LibConst.U8_MAX;
u8gTTC580Version_Major.CanMin :=VBasic.LibConst.U8_MIN;
u8gTTC580Version_Major.CanUnit :="";
u8gTTC580Version_Major.Description :="Program Version Major C0 TTC580";
u8gTTC580Version_Major.ErrorReaction := eErrorReaction.ERSIG_DFLT;
u8gTTC580Version_Major.ReceiverAdress :=1;
u8gTTC580Version_Major.ToolScalingDivisor :=1;
u8gTTC580Version_Major.ToolScalingMultiplier :=1;
u8gTTC580Version_Major.ToolScalingOffset :=0;
u8gTTC580Version_Major.ToolUnit :="";

u8gTTC580Version_Minor.AppScalingDivisor :=1;
u8gTTC580Version_Minor.AppScalingMultiplier :=1;
u8gTTC580Version_Minor.AppScalingOffset :=0;
u8gTTC580Version_Minor.AppUnit :="";
u8gTTC580Version_Minor.CanDefault :=0;
u8gTTC580Version_Minor.CanInit :=0;
u8gTTC580Version_Minor.CanMax :=VBasic.LibConst.U8_MAX;
u8gTTC580Version_Minor.CanMin :=VBasic.LibConst.U8_MIN;
u8gTTC580Version_Minor.CanUnit :="";
u8gTTC580Version_Minor.Description :="Program Version Minor C0 TTC580";
u8gTTC580Version_Minor.ErrorReaction := eErrorReaction.ERSIG_DFLT;
u8gTTC580Version_Minor.ReceiverAdress :=1;
u8gTTC580Version_Minor.ToolScalingDivisor :=1;
u8gTTC580Version_Minor.ToolScalingMultiplier :=1;
u8gTTC580Version_Minor.ToolScalingOffset :=0;
u8gTTC580Version_Minor.ToolUnit :="";

u8gTTC580Version_Patch.AppScalingDivisor :=1;
u8gTTC580Version_Patch.AppScalingMultiplier :=1;
u8gTTC580Version_Patch.AppScalingOffset :=0;
u8gTTC580Version_Patch.AppUnit :="";
u8gTTC580Version_Patch.CanDefault :=0;
u8gTTC580Version_Patch.CanInit :=0;
u8gTTC580Version_Patch.CanMax :=VBasic.LibConst.U8_MAX;
u8gTTC580Version_Patch.CanMin :=VBasic.LibConst.U8_MIN;
u8gTTC580Version_Patch.CanUnit :="";
u8gTTC580Version_Patch.Description :="Program Version Path C0 TTC580";
u8gTTC580Version_Patch.ErrorReaction := eErrorReaction.ERSIG_DFLT;
u8gTTC580Version_Patch.ReceiverAdress :=1;
u8gTTC580Version_Patch.ToolScalingDivisor :=1;
u8gTTC580Version_Patch.ToolScalingMultiplier :=1;
u8gTTC580Version_Patch.ToolScalingOffset :=0;
u8gTTC580Version_Patch.ToolUnit :="";

u8gTTC580Version_Custom.AppScalingDivisor :=1;
u8gTTC580Version_Custom.AppScalingMultiplier :=1;
u8gTTC580Version_Custom.AppScalingOffset :=0;
u8gTTC580Version_Custom.AppUnit :="";
u8gTTC580Version_Custom.CanDefault :=0;
u8gTTC580Version_Custom.CanInit :=0;
u8gTTC580Version_Custom.CanMax :=VBasic.LibConst.U8_MAX;
u8gTTC580Version_Custom.CanMin :=VBasic.LibConst.U8_MIN;
u8gTTC580Version_Custom.CanUnit :="";
u8gTTC580Version_Custom.Description :="Program Version Custom C0 TTC580";
u8gTTC580Version_Custom.ErrorReaction := eErrorReaction.ERSIG_DFLT;
u8gTTC580Version_Custom.ReceiverAdress :=1;
u8gTTC580Version_Custom.ToolScalingDivisor :=1;
u8gTTC580Version_Custom.ToolScalingMultiplier :=1;
u8gTTC580Version_Custom.ToolScalingOffset :=0;
u8gTTC580Version_Custom.ToolUnit :="";

i16gJoystAdvanceScaling.AppScalingDivisor :=1;
i16gJoystAdvanceScaling.AppScalingMultiplier :=1;
i16gJoystAdvanceScaling.AppScalingOffset :=0;
i16gJoystAdvanceScaling.AppUnit :="";
i16gJoystAdvanceScaling.CanDefault :=0;
i16gJoystAdvanceScaling.CanInit :=0;
i16gJoystAdvanceScaling.CanMax :=VBasic.LibConst.I16_MAX;
i16gJoystAdvanceScaling.CanMin :=VBasic.LibConst.I16_MIN;
i16gJoystAdvanceScaling.CanUnit :="";
i16gJoystAdvanceScaling.Description :="Joystick Advance Scaling Value";
i16gJoystAdvanceScaling.ErrorReaction := eErrorReaction.ERSIG_DFLT;
i16gJoystAdvanceScaling.ReceiverAdress :=1;
i16gJoystAdvanceScaling.ToolScalingDivisor :=1;
i16gJoystAdvanceScaling.ToolScalingMultiplier :=1;
i16gJoystAdvanceScaling.ToolScalingOffset :=0;
i16gJoystAdvanceScaling.ToolUnit :="";


                
END_METHOD
END_FUNCTION_BLOCK

FUNCTION_BLOCK Msg11C0SendToEvision7MessageClass EXTENDS CanReceiveMessageClass
  VAR_INPUT
    i16gSlopeLongAngle : Int16CanSignalClass;
    i16gSlopeTransAngle : Int16CanSignalClass;
    i16gSlopeResultAngle : Int16CanSignalClass;
    i16gTemperatureTransmissionValue : Int16CanSignalClass;
    Counter : UInt32CanSignalClass;
  END_VAR

            
          

METHOD SetData
  VAR_INPUT
    CanMsgPointer : POINTER TO CanMessageClass;
  END_VAR
                  IF IsValidPointer(canMsgPointer,'SetData') THEN
	SUPER^.SetData(CanMsgPointer);
	//Set the new data
	i16gSlopeLongAngle.Value := canMsgPointer^.GetInt16(0);
	i16gSlopeTransAngle.Value := canMsgPointer^.GetInt16(16);
	i16gSlopeResultAngle.Value := canMsgPointer^.GetInt16(32);
	i16gTemperatureTransmissionValue.Value := canMsgPointer^.GetInt16(48);
	//And increase the counter
	Counter.Value := CanMsgPointer^.Counter.Value;
END_IF

                
END_METHOD

PROPERTY i16gSlopeLongAngleRawValue : INT
GET
                    IF i16gSlopeLongAngle.AppScalingMultiplier = 0 THEN
	_MatchLog^.Error("Get i16gSlopeLongAngleRawValue", "Division by Zero!");
	RETURN;
End_IF

i16gSlopeLongAngleRawValue := TO_INT((i16gSlopeLongAngle.Value - i16gSlopeLongAngle.AppScalingOffset) * i16gSlopeLongAngle.AppScalingDivisor / i16gSlopeLongAngle.AppScalingMultiplier);

                  
END_GET
END_PROPERTY

PROPERTY i16gSlopeTransAngleRawValue : INT
GET
                    IF i16gSlopeTransAngle.AppScalingMultiplier = 0 THEN
	_MatchLog^.Error("Get i16gSlopeTransAngleRawValue", "Division by Zero!");
	RETURN;
End_IF

i16gSlopeTransAngleRawValue := TO_INT((i16gSlopeTransAngle.Value - i16gSlopeTransAngle.AppScalingOffset) * i16gSlopeTransAngle.AppScalingDivisor / i16gSlopeTransAngle.AppScalingMultiplier);

                  
END_GET
END_PROPERTY

PROPERTY i16gSlopeResultAngleRawValue : INT
GET
                    IF i16gSlopeResultAngle.AppScalingMultiplier = 0 THEN
	_MatchLog^.Error("Get i16gSlopeResultAngleRawValue", "Division by Zero!");
	RETURN;
End_IF

i16gSlopeResultAngleRawValue := TO_INT((i16gSlopeResultAngle.Value - i16gSlopeResultAngle.AppScalingOffset) * i16gSlopeResultAngle.AppScalingDivisor / i16gSlopeResultAngle.AppScalingMultiplier);

                  
END_GET
END_PROPERTY

PROPERTY i16gTemperatureTransmissionValueRawValue : INT
GET
                    IF i16gTemperatureTransmissionValue.AppScalingMultiplier = 0 THEN
	_MatchLog^.Error("Get i16gTemperatureTransmissionValueRawValue", "Division by Zero!");
	RETURN;
End_IF

i16gTemperatureTransmissionValueRawValue := TO_INT((i16gTemperatureTransmissionValue.Value - i16gTemperatureTransmissionValue.AppScalingOffset) * i16gTemperatureTransmissionValue.AppScalingDivisor / i16gTemperatureTransmissionValue.AppScalingMultiplier);

                  
END_GET
END_PROPERTY

PROPERTY i16gSlopeLongAngleToolValue : INT
GET
                    IF i16gSlopeLongAngle.ToolScalingDivisor = 0 OR i16gSlopeLongAngle.AppScalingMultiplier = 0 THEN
	_MatchLog^.Error("Get i16gSlopeLongAngleToolValue", "Division by Zero!");
	RETURN;
END_IF

i16gSlopeLongAngleToolValue := TO_INT(((i16gSlopeLongAngle.Value - i16gSlopeLongAngle.AppScalingOffset) * i16gSlopeLongAngle.AppScalingDivisor / i16gSlopeLongAngle.AppScalingMultiplier * i16gSlopeLongAngle.ToolScalingMultiplier / i16gSlopeLongAngle.ToolScalingDivisor) + i16gSlopeLongAngle.ToolScalingOffset);

                  
END_GET
END_PROPERTY

PROPERTY i16gSlopeTransAngleToolValue : INT
GET
                    IF i16gSlopeTransAngle.ToolScalingDivisor = 0 OR i16gSlopeTransAngle.AppScalingMultiplier = 0 THEN
	_MatchLog^.Error("Get i16gSlopeTransAngleToolValue", "Division by Zero!");
	RETURN;
END_IF

i16gSlopeTransAngleToolValue := TO_INT(((i16gSlopeTransAngle.Value - i16gSlopeTransAngle.AppScalingOffset) * i16gSlopeTransAngle.AppScalingDivisor / i16gSlopeTransAngle.AppScalingMultiplier * i16gSlopeTransAngle.ToolScalingMultiplier / i16gSlopeTransAngle.ToolScalingDivisor) + i16gSlopeTransAngle.ToolScalingOffset);

                  
END_GET
END_PROPERTY

PROPERTY i16gSlopeResultAngleToolValue : INT
GET
                    IF i16gSlopeResultAngle.ToolScalingDivisor = 0 OR i16gSlopeResultAngle.AppScalingMultiplier = 0 THEN
	_MatchLog^.Error("Get i16gSlopeResultAngleToolValue", "Division by Zero!");
	RETURN;
END_IF

i16gSlopeResultAngleToolValue := TO_INT(((i16gSlopeResultAngle.Value - i16gSlopeResultAngle.AppScalingOffset) * i16gSlopeResultAngle.AppScalingDivisor / i16gSlopeResultAngle.AppScalingMultiplier * i16gSlopeResultAngle.ToolScalingMultiplier / i16gSlopeResultAngle.ToolScalingDivisor) + i16gSlopeResultAngle.ToolScalingOffset);

                  
END_GET
END_PROPERTY

PROPERTY i16gTemperatureTransmissionValueToolValue : INT
GET
                    IF i16gTemperatureTransmissionValue.ToolScalingDivisor = 0 OR i16gTemperatureTransmissionValue.AppScalingMultiplier = 0 THEN
	_MatchLog^.Error("Get i16gTemperatureTransmissionValueToolValue", "Division by Zero!");
	RETURN;
END_IF

i16gTemperatureTransmissionValueToolValue := TO_INT(((i16gTemperatureTransmissionValue.Value - i16gTemperatureTransmissionValue.AppScalingOffset) * i16gTemperatureTransmissionValue.AppScalingDivisor / i16gTemperatureTransmissionValue.AppScalingMultiplier * i16gTemperatureTransmissionValue.ToolScalingMultiplier / i16gTemperatureTransmissionValue.ToolScalingDivisor) + i16gTemperatureTransmissionValue.ToolScalingOffset);

                  
END_GET
END_PROPERTY

METHOD InitializeCanSignals
                  i16gSlopeLongAngle.AppScalingDivisor :=1;
i16gSlopeLongAngle.AppScalingMultiplier :=1;
i16gSlopeLongAngle.AppScalingOffset :=0;
i16gSlopeLongAngle.AppUnit :="";
i16gSlopeLongAngle.CanDefault :=0;
i16gSlopeLongAngle.CanInit :=0;
i16gSlopeLongAngle.CanMax :=VBasic.LibConst.I16_MAX;
i16gSlopeLongAngle.CanMin :=VBasic.LibConst.I16_MIN;
i16gSlopeLongAngle.CanUnit :="";
i16gSlopeLongAngle.Description :="Slope Longitudinal Angle";
i16gSlopeLongAngle.ErrorReaction := eErrorReaction.ERSIG_DFLT;
i16gSlopeLongAngle.ReceiverAdress :=1;
i16gSlopeLongAngle.ToolScalingDivisor :=1;
i16gSlopeLongAngle.ToolScalingMultiplier :=1;
i16gSlopeLongAngle.ToolScalingOffset :=0;
i16gSlopeLongAngle.ToolUnit :="";

i16gSlopeTransAngle.AppScalingDivisor :=1;
i16gSlopeTransAngle.AppScalingMultiplier :=1;
i16gSlopeTransAngle.AppScalingOffset :=0;
i16gSlopeTransAngle.AppUnit :="";
i16gSlopeTransAngle.CanDefault :=0;
i16gSlopeTransAngle.CanInit :=0;
i16gSlopeTransAngle.CanMax :=VBasic.LibConst.I16_MAX;
i16gSlopeTransAngle.CanMin :=VBasic.LibConst.I16_MIN;
i16gSlopeTransAngle.CanUnit :="";
i16gSlopeTransAngle.Description :="Slope Transversal Angle";
i16gSlopeTransAngle.ErrorReaction := eErrorReaction.ERSIG_DFLT;
i16gSlopeTransAngle.ReceiverAdress :=1;
i16gSlopeTransAngle.ToolScalingDivisor :=1;
i16gSlopeTransAngle.ToolScalingMultiplier :=1;
i16gSlopeTransAngle.ToolScalingOffset :=0;
i16gSlopeTransAngle.ToolUnit :="";

i16gSlopeResultAngle.AppScalingDivisor :=1;
i16gSlopeResultAngle.AppScalingMultiplier :=1;
i16gSlopeResultAngle.AppScalingOffset :=0;
i16gSlopeResultAngle.AppUnit :="";
i16gSlopeResultAngle.CanDefault :=0;
i16gSlopeResultAngle.CanInit :=0;
i16gSlopeResultAngle.CanMax :=VBasic.LibConst.I16_MAX;
i16gSlopeResultAngle.CanMin :=VBasic.LibConst.I16_MIN;
i16gSlopeResultAngle.CanUnit :="";
i16gSlopeResultAngle.Description :="Slope Result Angle";
i16gSlopeResultAngle.ErrorReaction := eErrorReaction.ERSIG_DFLT;
i16gSlopeResultAngle.ReceiverAdress :=1;
i16gSlopeResultAngle.ToolScalingDivisor :=1;
i16gSlopeResultAngle.ToolScalingMultiplier :=1;
i16gSlopeResultAngle.ToolScalingOffset :=0;
i16gSlopeResultAngle.ToolUnit :="";

i16gTemperatureTransmissionValue.AppScalingDivisor :=1;
i16gTemperatureTransmissionValue.AppScalingMultiplier :=1;
i16gTemperatureTransmissionValue.AppScalingOffset :=0;
i16gTemperatureTransmissionValue.AppUnit :="";
i16gTemperatureTransmissionValue.CanDefault :=0;
i16gTemperatureTransmissionValue.CanInit :=0;
i16gTemperatureTransmissionValue.CanMax :=VBasic.LibConst.I16_MAX;
i16gTemperatureTransmissionValue.CanMin :=VBasic.LibConst.I16_MIN;
i16gTemperatureTransmissionValue.CanUnit :="";
i16gTemperatureTransmissionValue.Description :="Temp. Transmission value";
i16gTemperatureTransmissionValue.ErrorReaction := eErrorReaction.ERSIG_DFLT;
i16gTemperatureTransmissionValue.ReceiverAdress :=1;
i16gTemperatureTransmissionValue.ToolScalingDivisor :=1;
i16gTemperatureTransmissionValue.ToolScalingMultiplier :=1;
i16gTemperatureTransmissionValue.ToolScalingOffset :=0;
i16gTemperatureTransmissionValue.ToolUnit :="";


                
END_METHOD
END_FUNCTION_BLOCK

FUNCTION_BLOCK Msg12C0SendToEvision7MessageClass EXTENDS CanReceiveMessageClass
  VAR_INPUT
    i32gDistanceTraveledMeasureMast : Int32CanSignalClass;
    u32gTotalDistance : UInt32CanSignalClass;
    Counter : UInt32CanSignalClass;
  END_VAR

            
          

METHOD SetData
  VAR_INPUT
    CanMsgPointer : POINTER TO CanMessageClass;
  END_VAR
                  IF IsValidPointer(canMsgPointer,'SetData') THEN
	SUPER^.SetData(CanMsgPointer);
	//Set the new data
	i32gDistanceTraveledMeasureMast.Value := canMsgPointer^.GetInt32(0);
	u32gTotalDistance.Value := canMsgPointer^.GetUint32(32);
	//And increase the counter
	Counter.Value := CanMsgPointer^.Counter.Value;
END_IF

                
END_METHOD

PROPERTY i32gDistanceTraveledMeasureMastRawValue : DINT
GET
                    IF i32gDistanceTraveledMeasureMast.AppScalingMultiplier = 0 THEN
	_MatchLog^.Error("Get i32gDistanceTraveledMeasureMastRawValue", "Division by Zero!");
	RETURN;
End_IF

i32gDistanceTraveledMeasureMastRawValue := TO_DINT((i32gDistanceTraveledMeasureMast.Value - i32gDistanceTraveledMeasureMast.AppScalingOffset) * i32gDistanceTraveledMeasureMast.AppScalingDivisor / i32gDistanceTraveledMeasureMast.AppScalingMultiplier);

                  
END_GET
END_PROPERTY

PROPERTY u32gTotalDistanceRawValue : UDINT
GET
                    IF u32gTotalDistance.AppScalingMultiplier = 0 THEN
	_MatchLog^.Error("Get u32gTotalDistanceRawValue", "Division by Zero!");
	RETURN;
End_IF

